// TwinCAT 3 PLC project Untitled1
// ProgramVersion: 3.1.4026.25
// libraries:
//   Tc2_Standard, * (Beckhoff Automation GmbH)
//   Tc2_EtherCAT, * (Beckhoff Automation GmbH)
//   Tc2_System, * (Beckhoff Automation GmbH)
//   Festo_VTEM_DevCon,3.5.7.237,Festo SE & Co. KG
// project tree:
//   / PlcTask.TcTTO
//   POUs/ MAIN.TcPOU, FB_TandemConveyor.TcPOU, FB_CsvDriveSettings.TcPOU
// real-time tasks:
//   TASK PlcTask: cycle T#1ms, priority 20, ADS port 350
// I/O:
//   DEVICE Gerät 1 (EtherCAT), AmsNetId 192.168.178.10.2.1
//     Term 1 (EK1100) [EK1100 EtherCAT Coupler (2A E-Bus)]
//       Term 2 (EL2008) [EL2008 8Ch. Dig. Output 24V, 0.5A]
//       Term 3 (EL2008) [EL2008 8Ch. Dig. Output 24V, 0.5A]
//       Term 4 (EL2004) [EL2004 4Ch. Dig. Output 24V, 0.5A]
//       Term 11 (EL2004) [EL2004 4Ch. Dig. Output 24V, 0.5A]
//       Term 12 (EL1018) [EL1018 8Ch. Dig. Input 24V, 10µs]
//       Term 13 (EL1014-0010) [EL1014-0010 4Ch. Dig. Input 24V, isolated, 10µs]
//       Term 14 (EL3068) [EL3068 8Ch. Ana. Input 0-10V]
//       Term 15 (EL7047) [EL7047 1Ch. Stepper motor output stage (50V, 5A)]
//       Term 22 (EL9011) [EL9011 End Terminal]
//   DEVICE Gerät 2 (EtherCAT), AmsNetId 192.168.178.10.3.1
//     Box 5 (CPX-FB38 64Byte) [CPX-FB38 EtherCAT Busmodul]
//   DEVICE Device 3 (EtherCAT), AmsNetId 10.145.4.14.4.1
//     Term 6 (EK1100) [EK1100 EtherCAT Coupler (2A E-Bus)]
//       Term 7 (EL7201-0010) [EL7201-0010 1Ch. MDP742 Servo motor output stage with OCT (50V, 2.8A RMS)]
//       Term 3 (EL9011) [EL9011 End Terminal]
// variable links:
//   Untitled1/Untitled1 Instance <-> Device 1 (EtherCAT)/Term 1 (EK1100)/Term 11 (EL2004)
//     PlcTask Outputs/MAIN.OpenValve{21..24} <-> Channel {1..4}/Output  (4 links)
//   Untitled1/Untitled1 Instance <-> Device 1 (EtherCAT)/Term 1 (EK1100)/Term 12 (EL1018)
//     PlcTask Inputs/MAIN.LightBarrierOn{1..8} <-> Channel {1..8}/Input  (8 links)
//   Untitled1/Untitled1 Instance <-> Device 1 (EtherCAT)/Term 1 (EK1100)/Term 14 (EL3068)
//     PlcTask Inputs/MAIN.RawNozzlePressure <-> AI Standard Channel 1/Value
//     PlcTask Inputs/MAIN.RawNozzlePressure2 <-> AI Standard Channel 2/Value
//   Untitled1/Untitled1 Instance <-> Device 1 (EtherCAT)/Term 1 (EK1100)/Term 2 (EL2008)
//     PlcTask Outputs/MAIN.OpenValve{1..8} <-> Channel {1..8}/Output  (8 links)
//   Untitled1/Untitled1 Instance <-> Device 1 (EtherCAT)/Term 1 (EK1100)/Term 3 (EL2008)
//     PlcTask Outputs/MAIN.OpenValve{9..16} <-> Channel {1..8}/Output  (8 links)
//   Untitled1/Untitled1 Instance <-> Device 1 (EtherCAT)/Term 1 (EK1100)/Term 4 (EL2004)
//     PlcTask Outputs/MAIN.OpenValve{17..20} <-> Channel {1..4}/Output  (4 links)
//   Untitled1/Untitled1 Instance <-> Device 2 (EtherCAT)/Box 5 (CPX-FB38 64Byte)
//     PlcTask Inputs/MAIN.Valve0_IN[0] @bit 8 <-> Inputs/IB1
//     PlcTask Inputs/MAIN.Valve0_IN[1] @bit 8 <-> Inputs/IB3
//     PlcTask Inputs/MAIN.Valve0_IN[2] @bit 8 <-> Inputs/IB5
//     PlcTask Inputs/MAIN.Valve1_IN[0] @bit 8 <-> Inputs/IB7
//     PlcTask Inputs/MAIN.Valve1_IN[1] @bit 8 <-> Inputs/IB9
//     PlcTask Inputs/MAIN.Valve1_IN[2] @bit 8 <-> Inputs/IB11
//     PlcTask Inputs/MAIN.Valve0_IN[0] <-> Inputs/MAIN.Valve0_IN[0]
//     PlcTask Inputs/MAIN.Valve0_IN[1] <-> Inputs/MAIN.Valve0_IN[1]
//     PlcTask Inputs/MAIN.Valve0_IN[2] <-> Inputs/MAIN.Valve0_IN[2]
//     PlcTask Inputs/MAIN.Valve1_IN[0] <-> Inputs/MAIN.Valve1_IN[0]
//     PlcTask Inputs/MAIN.Valve1_IN[1] <-> Inputs/MAIN.Valve1_IN[1]
//     PlcTask Inputs/MAIN.Valve1_IN[2] <-> Inputs/MAIN.Valve1_IN[2]
//     PlcTask Outputs/MAIN.Valve0_OUT[0] <-> Outputs/MAIN.Valve0_OUT[0]
//     PlcTask Outputs/MAIN.Valve0_OUT[1] <-> Outputs/MAIN.Valve0_OUT[1]
//     PlcTask Outputs/MAIN.Valve0_OUT[2] <-> Outputs/MAIN.Valve0_OUT[2]
//     PlcTask Outputs/MAIN.Valve1_OUT[0] <-> Outputs/MAIN.Valve1_OUT[0]
//     PlcTask Outputs/MAIN.Valve1_OUT[1] <-> Outputs/MAIN.Valve1_OUT[1]
//     PlcTask Outputs/MAIN.Valve1_OUT[2] <-> Outputs/MAIN.Valve1_OUT[2]
//     PlcTask Outputs/MAIN.Valve0_OUT[0] @bit 8 <-> Outputs/QB1
//     PlcTask Outputs/MAIN.Valve0_OUT[1] @bit 8 <-> Outputs/QB3
//     PlcTask Outputs/MAIN.Valve0_OUT[2] @bit 8 <-> Outputs/QB5
//     PlcTask Outputs/MAIN.Valve1_OUT[0] @bit 8 <-> Outputs/QB7
//     PlcTask Outputs/MAIN.Valve1_OUT[1] @bit 8 <-> Outputs/QB9
//     PlcTask Outputs/MAIN.Valve1_OUT[2] @bit 8 <-> Outputs/QB11
//   Untitled1/Untitled1 Instance <-> Device 3 (EtherCAT)/Term 6 (EK1100)/Term 7 (EL7201-0010)
//     PlcTask Inputs/MAIN.ConveyorServo1ActualVelocity <-> DRV Velocity actual value/Velocity actual value
//     PlcTask Inputs/MAIN.ConveyorServo1FeedbackInvalid <-> FB Status/Status/TxPDO State
//     PlcTask Inputs/MAIN.ConveyorServo1InfoState <-> InfoData/State
//     PlcTask Inputs/MAIN.ConveyorServo1Position <-> FB Position/Position
//     PlcTask Inputs/MAIN.ConveyorServo1Statusword <-> DRV Statusword/Statusword
//     PlcTask Inputs/MAIN.ConveyorServo1WcState <-> WcState/WcState
//     PlcTask Outputs/MAIN.ConveyorServo1Controlword <-> DRV Controlword/Controlword
//     PlcTask Outputs/MAIN.ConveyorServo1TargetVelocity <-> DRV Target velocity/Target velocity

CONFIGURATION Untitled1
    RESOURCE PLC ON TwinCAT3
        TASK PlcTask(INTERVAL := T#1ms, PRIORITY := 20);
        PROGRAM MAIN WITH PlcTask : MAIN;
    END_RESOURCE
END_CONFIGURATION

// ---- POUs/MAIN.TcPOU
PROGRAM MAIN
VAR
	State					: INT  := 0; //state machine to control valves and motion terminal
	State2					: INT  := 2; //state machine for nozzle array 2
	State3					: INT  := 0; //state machine for nozzle array 3 and second VTEM unit
	State4					: INT  := 2; //state machine for nozzle array 4
	Counter					: INT  := 0; //timer counter that is in multiples of the PLC task time
	Counter2				: INT  := 0; //timer counter for the second nozzle array
	Counter3				: INT  := 0;
	Counter4				: INT  := 0;
	ShotDurationCycles		: INT  := 100; //100 cycles at 1 ms task time = 100 ms nozzle impulse
	ShotDurationCycles2		: INT  := 100; //pulse duration for the second nozzle array
	ShotDurationCycles3		: INT  := 100;
	ShotDurationCycles4		: INT  := 100;
	DelayDurationCycles		: INT  := 0; //delay cycles at 1 ms task time
	DelayDurationCycles2	: INT  := 0; //delay cycles for the second nozzle array
	DelayDurationCycles3	: INT  := 0;
	DelayDurationCycles4	: INT  := 0;
	OffsetDelayCycles1		: INT  := 0; //velocity-derived delay cycles for the first nozzle array
	OffsetDelayCycles2		: INT  := 0; //velocity-derived delay cycles for the second nozzle array
	OffsetDelayCycles3		: INT  := 0;
	OffsetDelayCycles4		: INT  := 0;
	LatchedDelayCycles1		: INT  := 0;
	LatchedDelayCycles2		: INT  := 0;
	LatchedDelayCycles3		: INT  := 0;
	LatchedDelayCycles4		: INT  := 0;
	LatchedNozzleEndCycles1	: INT  := 100;
	LatchedNozzleEndCycles2	: INT  := 100;
	LatchedNozzleEndCycles3	: INT  := 100;
	LatchedNozzleEndCycles4	: INT  := 100;
	
	TimeDelay				: BOOL := 0;
	DelayCounter			: INT  := 0;
	DelayCounter2			: INT  := 0;
	VelocityTimer			: TON;
	VelocityTimer2			: TON;
	VelocityTimer3			: TON;
	VelocityTimer4			: TON;
	LastVelocityTimeMs		: INT  := 0;
	LastVelocityTime2Ms		: INT  := 0;
	LastVelocityTime3Ms		: INT  := 0;
	LastVelocityTime4Ms		: INT  := 0;
	VelocityTimingActive	: BOOL := FALSE;
	VelocityTiming2Active	: BOOL := FALSE;
	VelocityTiming3Active	: BOOL := FALSE;
	VelocityTiming4Active	: BOOL := FALSE;
	VelocityMeasurementValid: BOOL := FALSE;
	VelocityMeasurement2Valid: BOOL := FALSE;
	VelocityMeasurement3Valid: BOOL := FALSE;
	VelocityMeasurement4Valid: BOOL := FALSE;

	//GUI control values written through ADS
	GuiPressureMbar1		: INT  := 0; // GUI/profile supplies pressure after a PLC restart
	GuiPressureMbar2		: INT  := 0;
	GuiPressureMbar3		: INT  := 0;
	GuiPressureMbar4		: INT  := 0;
	GuiDelayMs1				: UINT := 0;
	GuiDelayMs2				: UINT := 0;
	GuiDelayMs3				: UINT := 0;
	GuiDelayMs4				: UINT := 0;
	GuiPulseDurationMs1		: UINT := 100;
	GuiPulseDurationMs2		: UINT := 100;
	GuiPulseDurationMs3		: UINT := 100;
	GuiPulseDurationMs4		: UINT := 100;
	GuiArrayEnabled1		: BOOL := FALSE; // GUI must explicitly arm nozzle arrays after a PLC restart
	GuiArrayEnabled2		: BOOL := FALSE;
	GuiArrayEnabled3		: BOOL := FALSE;
	GuiArrayEnabled4		: BOOL := FALSE;
	GuiNozzleEnabled1		: BOOL := TRUE;
	GuiNozzleEnabled2		: BOOL := TRUE;
	GuiNozzleEnabled3		: BOOL := TRUE;
	GuiNozzleEnabled4		: BOOL := TRUE;
	GuiNozzleEnabled5		: BOOL := FALSE;
	GuiNozzleEnabled6		: BOOL := FALSE;
	GuiNozzleEnabled7		: BOOL := TRUE;
	GuiNozzleEnabled8		: BOOL := TRUE;
	GuiNozzleEnabled9		: BOOL := TRUE;
	GuiNozzleEnabled10		: BOOL := TRUE;
	GuiNozzleEnabled11		: BOOL := FALSE;
	GuiNozzleEnabled12		: BOOL := FALSE;
	GuiNozzleEnabled13		: BOOL := TRUE;
	GuiNozzleEnabled14		: BOOL := TRUE;
	GuiNozzleEnabled15		: BOOL := TRUE;
	GuiNozzleEnabled16		: BOOL := TRUE;
	GuiNozzleEnabled17		: BOOL := FALSE;
	GuiNozzleEnabled18		: BOOL := FALSE;
	GuiNozzleEnabled19		: BOOL := TRUE;
	GuiNozzleEnabled20		: BOOL := TRUE;
	GuiNozzleEnabled21		: BOOL := TRUE;
	GuiNozzleEnabled22		: BOOL := TRUE;
	GuiNozzleEnabled23		: BOOL := FALSE;
	GuiNozzleEnabled24		: BOOL := FALSE;
	GuiResetVelocityEstimates	: BOOL := FALSE;
	GuiSensorSpacing12Mm	: REAL := 40.0;
	GuiSensorSpacing23Mm	: REAL := 196.0;
	GuiSensorSpacing34Mm	: REAL := 40.0;
	GuiSensorSpacing45Mm	: REAL := 196.0;
	GuiSensorSpacing56Mm	: REAL := 40.0;
	GuiSensorSpacing67Mm	: REAL := 196.0;
	GuiSensorSpacing78Mm	: REAL := 40.0;
	GuiSensor2ToArray1SpacingMm	: REAL := 50.0;
	GuiSensor4ToArray2SpacingMm	: REAL := 45.0;
	GuiSensor6ToArray3SpacingMm	: REAL := 45.0;
	GuiSensor8ToArray4SpacingMm	: REAL := 48.0;
	GuiConveyorEnabled		: BOOL := FALSE;
	GuiVelocityCheckMode	: BOOL := FALSE;
	GuiConveyorReverse		: BOOL := FALSE;
	GuiConveyorReset		: BOOL := FALSE;
	GuiConveyorSpeedMmPerSec	: REAL := 0.0;
	GuiConveyorMaxSpeedMmPerSec	: REAL := 1000.0;
	GuiConveyorCalibrationMode	: BOOL := FALSE;
	GuiCalibrationMarkerDistanceMm	: REAL := 315.0;
	GuiCalibrationJogSteps		: UDINT := 100;
	GuiCalibrationJogSpeedFullStepsPerSec	: REAL := 10.0;
	GuiCalibrationMoveLeft		: BOOL := FALSE;
	GuiCalibrationMoveRight		: BOOL := FALSE;
	GuiCalibrationCaptureLeftMark	: BOOL := FALSE;
	GuiCalibrationCaptureRightMark	: BOOL := FALSE;
	GuiCalibrationStop			: BOOL := FALSE;
	GuiConveyorMmPerFullStep	: REAL := 0.0;
	GuiConveyorCalibrationValid	: BOOL := FALSE;
	// Verified two AM8112 motors, direct drive, 50 mm rollers, same shaft direction.
	// Start remains an explicit GUI command; see CSVSaver/TANDEM_CONVEYOR.md.
	ConveyorServoCommissioned : BOOL := TRUE; // stationary setup and live CoE readback verified; GUI motion starts disabled
	ConveyorServoDirection1 : INT := 1; // same shaft direction, confirmed for the two 50 mm rollers
	ConveyorServoDirection2 : INT := 1;
	ConveyorServoMotor2Ratio : LREAL := 1.0; // motor 2 rev / motor 1 rev, including roller diameter
	ConveyorServoFeedbackCountsPerRev : LREAL := 1048576.0;
	ConveyorServoFeedbackCountsPerRev2 : LREAL := 1048576.0;
	ConveyorServoVelocityUnitsPerRevPerSec : LREAL := 268435.0; // live CoE 0x9010:14 readback
	ConveyorServoVelocityUnitsPerRevPerSec2 : LREAL := 268435.0;
	ConveyorServoMaxMotorRpm : LREAL := 5.0;
	ConveyorServoAccelerationRpmPerSec : LREAL := 5.0;
	ConveyorServoPositionGain : LREAL := 5.0;
	ConveyorServoSyncToleranceFullSteps : LREAL := 5.0;
	ConveyorServoFollowingToleranceFullSteps : LREAL := 20.0;
	// Authoritative NEW belt calibration: 200 virtual full steps per motor 1 revolution.
	// Legacy GUI profiles cannot overwrite this with the old stepper's scale.
	ConveyorServoCalibratedMmPerFullStep : REAL := 0.7853981634; // pi * 50 mm / 200; refine with GUI marker calibration
	ConveyorServoFaultCode : UINT := 0;
	ConveyorServoState : UINT := 0;
	ConveyorServoSyncErrorFullSteps : LREAL := 0.0;
	ConveyorServoStopRequested : BOOL := FALSE;
	ConveyorServoResetRequested : BOOL := FALSE;
	TandemConveyor : FB_TandemConveyor;
	ConveyorDriveSettings : FB_CsvDriveSettings;
	GuiOffsetMm1			: REAL := 0.0;
	GuiOffsetMm2			: REAL := 0.0;
	GuiOffsetMm3			: REAL := 0.0;
	GuiOffsetMm4			: REAL := 0.0;
	GuiForceDelayMeasurementEnabled	: BOOL := FALSE;
	GuiForceDelayLightBarrier	: UINT := 2;
	GuiForceDelaySensor		: UINT := 1;
	GuiForceDelayWindowMs		: UINT := 2000;
	GuiForceDelayMinRise		: REAL := 0.05;
	GuiForceDelayReset		: BOOL := FALSE;
	GuiForceResponseDelayMs1	: REAL := 8.7;
	GuiForceResponseDelayMs2	: REAL := 8.7;
	GuiForceResponseDelayMs3	: REAL := 8.7;
	GuiForceResponseDelayMs4	: REAL := 8.7;
	GuiForceSingleNozzleResponseDelayMs1	: REAL := 8.7;
	GuiForceSingleNozzleResponseDelayMs2	: REAL := 8.7;
	GuiForceSingleNozzleResponseDelayMs3	: REAL := 8.7;
	GuiForceSingleNozzleResponseDelayMs4	: REAL := 8.7;
	// BiBaZu Reorientation Control ADS contract
	GuiReorientationControlActive	: BOOL := FALSE;
	GuiReorientationHeartbeat		: UDINT := 0;
	GuiReorientationStart			: BOOL := FALSE;
	GuiReorientationAbort			: BOOL := FALSE;
	GuiReorientationReset			: BOOL := FALSE;
	GuiReorientationLegacyTakeover	: BOOL := FALSE;
	GuiReorientationExpectedArrayMask	: BYTE := 0;
	// Continuous production-run staging area.  The GUI writes every field first
	// and publishes it atomically by incrementing QueueCommit last.
	GuiReorientationFinish			: BOOL := FALSE;
	GuiReorientationResultAck		: UDINT := 0;
	GuiReorientationQueueCommit		: UDINT := 0;
	GuiReorientationQueueSequence	: UDINT := 0;
	GuiReorientationQueueTrackId		: UDINT := 0;
	GuiReorientationQueuePoseId		: UINT := 0;
	GuiReorientationQueueDecisionCode	: UINT := 0;
	GuiReorientationQueueArrayMask	: BYTE := 0;
	GuiReorientationQueueNozzleMask1	: BYTE := 0;
	GuiReorientationQueueNozzleMask2	: BYTE := 0;
	GuiReorientationQueueNozzleMask3	: BYTE := 0;
	GuiReorientationQueueNozzleMask4	: BYTE := 0;
	GuiReorientationQueuePressureMbar1	: INT := 0;
	GuiReorientationQueuePressureMbar2	: INT := 0;
	GuiReorientationQueuePressureMbar3	: INT := 0;
	GuiReorientationQueuePressureMbar4	: INT := 0;
	GuiReorientationQueueDelayMs1	: UINT := 0;
	GuiReorientationQueueDelayMs2	: UINT := 0;
	GuiReorientationQueueDelayMs3	: UINT := 0;
	GuiReorientationQueueDelayMs4	: UINT := 0;
	GuiReorientationQueuePulseMs1	: UINT := 1;
	GuiReorientationQueuePulseMs2	: UINT := 1;
	GuiReorientationQueuePulseMs3	: UINT := 1;
	GuiReorientationQueuePulseMs4	: UINT := 1;
	GuiReorientationQueueOffsetMm1	: REAL := 0.0;
	GuiReorientationQueueOffsetMm2	: REAL := 0.0;
	GuiReorientationQueueOffsetMm3	: REAL := 0.0;
	GuiReorientationQueueOffsetMm4	: REAL := 0.0;
	GuiReorientationQueueForceResponseMs1	: REAL := 0.0;
	GuiReorientationQueueForceResponseMs2	: REAL := 0.0;
	GuiReorientationQueueForceResponseMs3	: REAL := 0.0;
	GuiReorientationQueueForceResponseMs4	: REAL := 0.0;
	GuiReorientationQueueForceSingleMs1	: REAL := 0.0;
	GuiReorientationQueueForceSingleMs2	: REAL := 0.0;
	GuiReorientationQueueForceSingleMs3	: REAL := 0.0;
	GuiReorientationQueueForceSingleMs4	: REAL := 0.0;
	ReorientationHeartbeatAck		: UDINT := 0;
	ReorientationHeartbeatAlive	: BOOL := FALSE;
	ReorientationState				: UINT := 0; //0 legacy,10 armed,20 running,30 drain,40 complete,90+ fault
	ReorientationFaultCode			: UINT := 0;
	ReorientationBusy				: BOOL := FALSE;
	ReorientationExitSeen			: BOOL := FALSE;
	ReorientationArraysIdle		: BOOL := TRUE;
	ReorientationExpectedArrayMask	: BYTE := 0;
	ReorientationTriggeredArrayMask	: BYTE := 0;
	ReorientationComplete			: BOOL := FALSE;
	ReorientationCycleCounter		: UDINT := 0;
	ReorientationLastHeartbeat		: UDINT := 0;
	ReorientationHeartbeatAgeMs	: UDINT := 0;
	ReorientationCycleAgeMs		: UDINT := 0;
	ReorientationDrainAgeMs		: UDINT := 0;
	ReorientationSafeLatch			: BOOL := FALSE;
	// Diagnostic context retained for non-fatal light-barrier warnings and for
	// compatibility with older GUIs that reported these conditions as fault 96.
	ReorientationFaultDetail		: UINT := 0; // 1=no clear, 2=queue mismatch, 3=sensor order
	ReorientationFaultSensor		: UINT := 0;
	ReorientationFaultExpectedSequence	: UDINT := 0;
	ReorientationFaultPreviousSequence	: UDINT := 0;
	ReorientationFaultQueueAck		: UDINT := 0;
	ReorientationFaultQueueSlotSequence	: UDINT := 0;
	ReorientationFaultBarrierStableMask	: BYTE := 0;
	// Non-fatal resynchronization after an intentionally airborne workpiece
	// skips barriers downstream of its final active nozzle array.
	// 1=downstream barriers skipped, 2=airborne duplicate, 3=no-clear edge,
	// 4=edge without matching queue slot, 5=out-of-order edge. All are non-fatal.
	ReorientationWarningCode		: UINT := 0;
	ReorientationWarningSensor		: UINT := 0;
	ReorientationWarningSequence	: UDINT := 0;
	ReorientationWarningPreviousSequence	: UDINT := 0;
	ReorientationWarningSkippedBarrierMask	: BYTE := 0;
	ReorientationWarningCounter		: UDINT := 0;
	// Public continuous-run queue/result diagnostics.
	ReorientationQueueDepth			: UINT := 0;
	ReorientationQueueCapacity		: UINT := 128;
	ReorientationQueueEnqueueAck		: UDINT := 0;
	ReorientationQueueEnteredCount	: UDINT := 0;
	ReorientationQueueCompletedCount	: UDINT := 0;
	ReorientationQueueBypassCount		: UDINT := 0;
	ReorientationSensorSequence1	: UDINT := 0;
	ReorientationSensorSequence2	: UDINT := 0;
	ReorientationSensorSequence3	: UDINT := 0;
	ReorientationSensorSequence4	: UDINT := 0;
	ReorientationSensorSequence5	: UDINT := 0;
	ReorientationSensorSequence6	: UDINT := 0;
	ReorientationSensorSequence7	: UDINT := 0;
	ReorientationSensorSequence8	: UDINT := 0;
	ReorientationResultAvailable	: BOOL := FALSE;
	ReorientationResultSequence		: UDINT := 0;
	ReorientationResultTriggeredMask	: BYTE := 0;
	ReorientationResultFaultCode	: UINT := 0;
	// Frozen 128-part ring.  A slot is not reusable until its result is ACKed.
	BatchQueueSequence				: ARRAY [0..127] OF UDINT;
	BatchQueueTrackId				: ARRAY [0..127] OF UDINT;
	BatchQueuePoseId				: ARRAY [0..127] OF UINT;
	BatchQueueDecisionCode			: ARRAY [0..127] OF UINT;
	BatchQueueArrayMask				: ARRAY [0..127] OF BYTE;
	BatchQueueNozzleMask			: ARRAY [0..127, 1..4] OF BYTE;
	BatchQueuePressureMbar			: ARRAY [0..127, 1..4] OF INT;
	BatchQueueDelayMs				: ARRAY [0..127, 1..4] OF UINT;
	BatchQueuePulseMs				: ARRAY [0..127, 1..4] OF UINT;
	BatchQueueOffsetMm				: ARRAY [0..127, 1..4] OF REAL;
	BatchQueueForceResponseMs		: ARRAY [0..127, 1..4] OF REAL;
	BatchQueueForceSingleMs			: ARRAY [0..127, 1..4] OF REAL;
	BatchQueuePairStartMs			: ARRAY [0..127, 1..4] OF UDINT;
	BatchQueueTriggeredMask			: ARRAY [0..127] OF BYTE;
	// Unlike TriggeredMask, this is set only while a real valve output is
	// commanded open. It marks this exact queued part as eligible for flight
	// recovery; it cannot prove pneumatic pressure or actual part motion.
	BatchQueueActuatedMask			: ARRAY [0..127] OF BYTE;
	BatchQueueFinishedMask			: ARRAY [0..127] OF BYTE;
	BatchQueueExitSeen				: ARRAY [0..127] OF BOOL;
	BatchResultSequence				: ARRAY [0..127] OF UDINT;
	BatchResultTriggeredMask		: ARRAY [0..127] OF BYTE;
	BatchResultFaultCode			: ARRAY [0..127] OF UINT;
	BatchNextSensorSequence			: ARRAY [1..8] OF UDINT;
	BatchSensorSequence				: ARRAY [1..8] OF UDINT;
	BatchSensorFalling				: ARRAY [1..8] OF BOOL;
	BatchSensorStable				: ARRAY [1..8] OF BOOL;
	BatchPairSpacingMm				: ARRAY [1..4] OF REAL;
	BatchSensorToArraySpacingMm	: ARRAY [1..4] OF REAL;
	BatchSensorNeedsClear			: ARRAY [1..8] OF BOOL;
	PairedFirstBarrierFalling		: ARRAY [1..4] OF BOOL;
	PairedFirstBarrierLocked		: ARRAY [1..4] OF BOOL;
	PairedFirstBarrierLockStartMs	: ARRAY [1..4] OF UDINT;
	PairedSecondBarrierFalling		: ARRAY [1..4] OF BOOL;
	PairedSecondBarrierLocked		: ARRAY [1..4] OF BOOL;
	PairedSecondBarrierLockStartMs	: ARRAY [1..4] OF UDINT;
	PairedBarrierLockTimeoutMs		: UDINT := 500;
	BatchSensorOrderInvalid			: BOOL := FALSE;
	BatchCanResyncSkippedSensors	: BOOL := FALSE;
	BatchCurrentFlightConfirmed	: BOOL := FALSE;
	BatchIgnoreAirborneDuplicate	: BOOL := FALSE;
	BatchLastRequiredSensor			: INT := 0;
	BatchLastRequiredArrayMask		: BYTE := 0;
	BatchPreviousSlotIndex			: INT := 0;
	BatchPreviousLastRequiredSensor	: INT := 0;
	BatchPreviousLastRequiredArrayMask	: BYTE := 0;
	BatchResyncIndex					: INT := 0;
	BatchSkippedBarrierMask			: BYTE := 0;
	BatchCurrentBarrierStableMask	: BYTE := 0;
	BatchNextCompleteSequence		: UDINT := 1;
	BatchLastAcceptedCommit			: UDINT := 0;
	BatchAcceptedResultAck			: UDINT := 0;
	// Each array has its own 16-entry job FIFO.  Jobs contain the final delay,
	// pressure and nozzle mask and therefore remain immutable during a pulse.
	BatchJobSequence				: ARRAY [0..15, 1..4] OF UDINT;
	BatchJobNozzleMask				: ARRAY [0..15, 1..4] OF BYTE;
	BatchJobPressureMbar			: ARRAY [0..15, 1..4] OF INT;
	BatchJobDelayCycles				: ARRAY [0..15, 1..4] OF INT;
	BatchJobPulseCycles				: ARRAY [0..15, 1..4] OF INT;
	BatchJobHead					: ARRAY [1..4] OF UINT;
	BatchJobTail					: ARRAY [1..4] OF UINT;
	BatchJobCount					: ARRAY [1..4] OF UINT;
	BatchActiveSequence				: ARRAY [1..4] OF UDINT;
	BatchLoopIndex					: INT := 0;
	BatchSlotIndex					: INT := 0;
	BatchJobIndex					: INT := 0;
	BatchElapsedMs					: UDINT := 0;
	BatchComputedDelayMs			: REAL := 0.0;
	BatchResponseDelayMs			: REAL := 0.0;
	BatchNozzleCount				: INT := 0;
	EstimatedVelocityMmPerSec	: REAL := 0.0;
	EstimatedVelocityMmPerSec1	: REAL := 0.0;
	EstimatedVelocityMmPerSec2	: REAL := 0.0;
	EstimatedVelocityMmPerSec3	: REAL := 0.0;
	EstimatedVelocityMmPerSec4	: REAL := 0.0;
	EstimatedOffsetDelayMs1		: REAL := 0.0;
	EstimatedOffsetDelayMs2		: REAL := 0.0;
	EstimatedOffsetDelayMs3		: REAL := 0.0;
	EstimatedOffsetDelayMs4		: REAL := 0.0;
	Array1Active			: BOOL := FALSE;
	Array2Active			: BOOL := FALSE;
	Array3Active			: BOOL := FALSE;
	Array4Active			: BOOL := FALSE;
	ConveyorSpeedMmPerSec	: REAL := 0.0; //limited conveyor speed command in mm/s
	ConveyorVelocityRatio	: REAL := 0.0;
	ConveyorVelocityRaw		: INT := 0; //0..10000 legacy velocity command, adapted to both servos
	ConveyorFullStepsPerSec	: REAL := 0.0;
	ConveyorSpeedRangeFullStepsPerSec	: REAL := 2000.0; //legacy velocity scale, virtual full steps/s
	ConveyorMotionState		: INT := 0;
	ConveyorMotionMode		: INT := 0; //0 idle, 1 normal endless, 2 calibration move
	ConveyorActiveVelocity	: INT := 0;
	ConveyorActiveStartType	: UINT := 0;
	CalibrationTargetIncrements	: DINT := 0;
	CalibrationDirectionNegative	: BOOL := FALSE;
	CalibrationLeftMarkValid	: BOOL := FALSE;
	CalibrationRightMarkValid	: BOOL := FALSE;
	CalibrationLeftPosition		: UDINT := 0;
	CalibrationRightPosition	: UDINT := 0;
	CalibrationPositionDifferenceIncrements	: UDINT := 0;
	CalibrationFullStepDifference	: REAL := 0.0;
	CalibrationStepsPerMm		: REAL := 0.0;
	CalibrationBusy			: BOOL := FALSE;
	CalibrationError			: BOOL := FALSE;
	CalibrationStatusCode		: UINT := 0; //0 ready, 1 starting, 2 moving, 3 complete, 4 invalid, 5 drive error
	CalibrationPositionDelta	: LINT := 0;
	LastConveyorCalibrationMode	: BOOL := FALSE;
	GuiBarrierCalibrationFirstSensor	: UINT := 1;
	GuiBarrierCalibrationSecondSensor	: UINT := 2;
	GuiBarrierCalibrationDebounceMs	: UINT := 20;
	GuiLightBarrierInvert1	: BOOL := TRUE;
	GuiLightBarrierInvert2	: BOOL := TRUE;
	GuiLightBarrierInvert3	: BOOL := TRUE;
	GuiLightBarrierInvert4	: BOOL := TRUE;
	GuiLightBarrierInvert5	: BOOL := TRUE;
	GuiLightBarrierInvert6	: BOOL := TRUE;
	GuiLightBarrierInvert7	: BOOL := TRUE;
	GuiLightBarrierInvert8	: BOOL := TRUE;
	GuiLightBarrierDebounceEnabled1	: BOOL := FALSE;
	GuiLightBarrierDebounceEnabled2	: BOOL := FALSE;
	GuiLightBarrierDebounceEnabled3	: BOOL := FALSE;
	GuiLightBarrierDebounceEnabled4	: BOOL := FALSE;
	GuiLightBarrierDebounceEnabled5	: BOOL := FALSE;
	GuiLightBarrierDebounceEnabled6	: BOOL := FALSE;
	GuiLightBarrierDebounceEnabled7	: BOOL := FALSE;
	GuiLightBarrierDebounceEnabled8	: BOOL := FALSE;
	GuiBarrierCalibrationStart	: BOOL := FALSE;
	BarrierCalibrationActive	: BOOL := FALSE;
	BarrierCalibrationFirstCaptured	: BOOL := FALSE;
	BarrierCalibrationSecondCaptured	: BOOL := FALSE;
	BarrierCalibrationValid	: BOOL := FALSE;
	BarrierCalibrationFirstPosition	: UDINT := 0;
	BarrierCalibrationSecondPosition	: UDINT := 0;
	BarrierCalibrationDifferenceIncrements	: UDINT := 0;
	BarrierCalibrationDistanceMm	: REAL := 0.0;
	BarrierCalibrationPositionDelta	: LINT := 0;
	BarrierCalibrationFirstState	: BOOL := FALSE;
	BarrierCalibrationSecondState	: BOOL := FALSE;
	BarrierCalibrationFirstInitialState	: BOOL := FALSE;
	BarrierCalibrationSecondInitialState	: BOOL := FALSE;
	BarrierCalibrationFirstCandidatePosition	: UDINT := 0;
	BarrierCalibrationSecondCandidatePosition	: UDINT := 0;
	BarrierCalibrationFirstStableCycles	: UINT := 0;
	BarrierCalibrationSecondStableCycles	: UINT := 0;
	BarrierCalibrationAbortRequested	: BOOL := FALSE;
	BarrierCalibrationStatusCode	: UINT := 0; //0 ready, 1 waiting first, 2 waiting second, 3 complete, 4 invalid/cancelled, 5 drive error

	//IO Variables
	//EL 1018
	LightBarrierOn1 AT %I*	: BOOL := 0; //1 when detecting a reflection
	LightBarrierOn2 AT %I*	: BOOL := 0; //1 when detecting a reflection
	LightBarrierOn3 AT %I*	: BOOL := 0; //1 when detecting a reflection
	LightBarrierOn4 AT %I*	: BOOL := 0; //1 when detecting a reflection
	LightBarrierOn5 AT %I*	: BOOL := 0; //1 when detecting a reflection
	LightBarrierOn6 AT %I*	: BOOL := 0; //1 when detecting a reflection
	LightBarrierOn7 AT %I*	: BOOL := 0; //1 when detecting a reflection
	LightBarrierOn8 AT %I*	: BOOL := 0; //1 when detecting a reflection
	LightBarrierLogical1	: BOOL := FALSE;
	LightBarrierLogical2	: BOOL := FALSE;
	LightBarrierLogical3	: BOOL := FALSE;
	LightBarrierLogical4	: BOOL := FALSE;
	LightBarrierLogical5	: BOOL := FALSE;
	LightBarrierLogical6	: BOOL := FALSE;
	LightBarrierLogical7	: BOOL := FALSE;
	LightBarrierLogical8	: BOOL := FALSE;
	LastLightBarrierInvert1	: BOOL := FALSE;
	LastLightBarrierInvert2	: BOOL := FALSE;
	LastLightBarrierInvert3	: BOOL := TRUE;
	LastLightBarrierInvert4	: BOOL := TRUE;
	LastLightBarrierInvert5	: BOOL := FALSE;
	LastLightBarrierInvert6	: BOOL := FALSE;
	LastLightBarrierInvert7	: BOOL := TRUE;
	LastLightBarrierInvert8	: BOOL := TRUE;
	LastLightBarrierDebounceEnabled1	: BOOL := TRUE;
	LastLightBarrierDebounceEnabled2	: BOOL := TRUE;
	LastLightBarrierDebounceEnabled3	: BOOL := FALSE;
	LastLightBarrierDebounceEnabled4	: BOOL := FALSE;
	LastLightBarrierDebounceEnabled5	: BOOL := TRUE;
	LastLightBarrierDebounceEnabled6	: BOOL := TRUE;
	LastLightBarrierDebounceEnabled7	: BOOL := FALSE;
	LastLightBarrierDebounceEnabled8	: BOOL := FALSE;
	LightBarrierStable1		: BOOL := FALSE;
	LightBarrierStable2		: BOOL := FALSE;
	LightBarrierStable3		: BOOL := FALSE;
	LightBarrierStable4		: BOOL := FALSE;
	LightBarrierStable5		: BOOL := FALSE;
	LightBarrierStable6		: BOOL := FALSE;
	LightBarrierStable7		: BOOL := FALSE;
	LightBarrierStable8		: BOOL := FALSE;
	LightBarrierStableCounter1	: UINT := 0;
	LightBarrierStableCounter2	: UINT := 0;
	LightBarrierStableCounter3	: UINT := 0;
	LightBarrierStableCounter4	: UINT := 0;
	LightBarrierStableCounter5	: UINT := 0;
	LightBarrierStableCounter6	: UINT := 0;
	LightBarrierStableCounter7	: UINT := 0;
	LightBarrierStableCounter8	: UINT := 0;
	LightBarrierDebounceInitialized	: BOOL := FALSE;
	LastLightBarrier1		: BOOL := FALSE; //previous debounced state
	LastLightBarrier2		: BOOL := FALSE; //previous debounced state
	LastLightBarrier3		: BOOL := FALSE; //previous debounced state
	LastLightBarrier4		: BOOL := FALSE; //previous debounced state
	LastLightBarrier5		: BOOL := FALSE; //previous debounced state
	LastLightBarrier6		: BOOL := FALSE; //previous debounced state
	LastLightBarrier7		: BOOL := FALSE; //previous debounced state
	LastLightBarrier8		: BOOL := FALSE; //previous debounced state
	LightBarrier1FallingEdge	: BOOL := FALSE;
	LightBarrier2FallingEdge	: BOOL := FALSE;
	LightBarrier3FallingEdge	: BOOL := FALSE;
	LightBarrier4FallingEdge	: BOOL := FALSE;
	LightBarrier5FallingEdge	: BOOL := FALSE;
	LightBarrier6FallingEdge	: BOOL := FALSE;
	LightBarrier7FallingEdge	: BOOL := FALSE;
	LightBarrier8FallingEdge	: BOOL := FALSE;
	LightBarrierEventClockMs	: UDINT := 0; //1 ms PLC task cycle counter
	// ADS diagnostic ring: version, sequence, clock, then 256 records
	// (sequence, timestamp_ms, sensor * 2 + stable_state). Never consumed by ADS.
	LightBarrierEventHistory : ARRAY[0..770] OF UDINT;
	LightBarrierHistorySlot : UDINT := 0;
	// Actual alternating-gate outputs used by velocity timing and array triggers.
	// Same ring layout, but code bit 0 is the accepted-edge BOOL (1 for one cycle).
	LightBarrierFilteredEventHistory : ARRAY[0..770] OF UDINT;
	LightBarrierFilteredSignal : ARRAY[1..8] OF BOOL;
	LastLightBarrierFilteredSignal : ARRAY[1..8] OF BOOL;
	LightBarrierFilteredSensor : INT;
	LightBarrierFilteredSlot : UDINT;
	LightBarrierEventCount1	: UDINT := 0;
	LightBarrierEventCount2	: UDINT := 0;
	LightBarrierEventCount3	: UDINT := 0;
	LightBarrierEventCount4	: UDINT := 0;
	LightBarrierEventCount5	: UDINT := 0;
	LightBarrierEventCount6	: UDINT := 0;
	LightBarrierEventCount7	: UDINT := 0;
	LightBarrierEventCount8	: UDINT := 0;
	LightBarrierLastEventTimeMs1	: UDINT := 0;
	LightBarrierLastEventTimeMs2	: UDINT := 0;
	LightBarrierLastEventTimeMs3	: UDINT := 0;
	LightBarrierLastEventTimeMs4	: UDINT := 0;
	LightBarrierLastEventTimeMs5	: UDINT := 0;
	LightBarrierLastEventTimeMs6	: UDINT := 0;
	LightBarrierLastEventTimeMs7	: UDINT := 0;
	LightBarrierLastEventTimeMs8	: UDINT := 0;
	LightBarrierLastEventPosition1	: UDINT := 0;
	LightBarrierLastEventPosition2	: UDINT := 0;
	LightBarrierLastEventPosition3	: UDINT := 0;
	LightBarrierLastEventPosition4	: UDINT := 0;
	LightBarrierLastEventPosition5	: UDINT := 0;
	LightBarrierLastEventPosition6	: UDINT := 0;
	LightBarrierLastEventPosition7	: UDINT := 0;
	LightBarrierLastEventPosition8	: UDINT := 0;
	Array1TriggerPending		: BOOL := FALSE;
	Array2TriggerPending		: BOOL := FALSE;
	Array3TriggerPending		: BOOL := FALSE;
	Array4TriggerPending		: BOOL := FALSE;
	ForceDelayBusy			: BOOL := FALSE;
	ForceDelayStatusCode		: UINT := 0; //0 disabled, 1 armed, 2 measuring, 3 valid, 4 no peak
	ForceDelayResultCounter		: UDINT := 0;
	ForceDelayValidCount		: UDINT := 0;
	ForceDelayInvalidCount		: UDINT := 0;
	ForceDelayLastValid		: BOOL := FALSE;
	ForceDelayLightBarrierTimeMs	: UDINT := 0;
	ForceDelayPeakTimeMs		: UDINT := 0;
	ForceDelayPeakDelayMs		: UDINT := 0;
	ForceDelayElapsedMs		: UINT := 0;
	ForceDelayBaseline		: REAL := 0.0;
	ForceDelayPeak			: REAL := 0.0;
	ForceDelayPeakRise		: REAL := 0.0;
	ForceDelayCurrentSignal		: REAL := 0.0;
	ForceDelayBaselineBuffer1	: ARRAY [0..49] OF REAL;
	ForceDelayBaselineBuffer2	: ARRAY [0..49] OF REAL;
	ForceDelayBaselineSum1		: REAL := 0.0;
	ForceDelayBaselineSum2		: REAL := 0.0;
	ForceDelayBaselineIndex		: UINT := 0;
	ForceDelayBaselineCount		: UINT := 0;
	ForceDelayTrigger		: BOOL := FALSE;
	ActiveNozzleCount1		: INT := 0;
	ActiveNozzleCount2		: INT := 0;
	ActiveNozzleCount3		: INT := 0;
	ActiveNozzleCount4		: INT := 0;
	EffectiveForceResponseDelayMs1	: REAL := 0.0;
	EffectiveForceResponseDelayMs2	: REAL := 0.0;
	EffectiveForceResponseDelayMs3	: REAL := 0.0;
	EffectiveForceResponseDelayMs4	: REAL := 0.0;
	
	//EL 3068
	RawNozzlePressure AT %I*: INT  := 0; //The raw analogue input reading from the EL3068 terminal (max 32767)
	NozzlePressure			: REAL := 0.0; //converted to pressure value in bar
	
	RawNozzlePressure2 AT %I*: INT := 0; //raw reading from the second pressure sensor
	NozzlePressure2          : REAL := 0.0; //converted to pressure value in bar
	
	
	//Digital valve outputs
	//0 to close valve 1 to open valve
	OpenValve1 AT %Q*		: BOOL := 0;
	OpenValve2 AT %Q*		: BOOL := 0;
	OpenValve3 AT %Q*		: BOOL := 0;
	OpenValve4 AT %Q*		: BOOL := 0;
	OpenValve5 AT %Q*		: BOOL := 0;
	OpenValve6 AT %Q*		: BOOL := 0;
	OpenValve7 AT %Q*		: BOOL := 0;
	OpenValve8 AT %Q*		: BOOL := 0;
	OpenValve9 AT %Q*		: BOOL := 0;
	OpenValve10 AT %Q*		: BOOL := 0;
	OpenValve11 AT %Q*		: BOOL := 0;
	OpenValve12 AT %Q*		: BOOL := 0;
	OpenValve13 AT %Q*		: BOOL := 0;
	OpenValve14 AT %Q*		: BOOL := 0;
	OpenValve15 AT %Q*		: BOOL := 0;
	OpenValve16 AT %Q*		: BOOL := 0;
	OpenValve17 AT %Q*		: BOOL := 0;
	OpenValve18 AT %Q*		: BOOL := 0;
	OpenValve19 AT %Q*		: BOOL := 0;
	OpenValve20 AT %Q*		: BOOL := 0;
	OpenValve21 AT %Q*		: BOOL := 0;
	OpenValve22 AT %Q*		: BOOL := 0;
	OpenValve23 AT %Q*		: BOOL := 0;
	OpenValve24 AT %Q*		: BOOL := 0;

	// Existing ADS contract, now backed by FB_TandemConveyor rather than EL7047 I/O.
	StepperStmStatus : WORD := 0;
	StepperPosBusy : BOOL := FALSE;
	StepperPosInTarget : BOOL := FALSE;
	StepperPosWarning : BOOL := FALSE;
	StepperPosError : BOOL := FALSE;
	StepperPosReadyToExecute : BOOL := FALSE;
	StepperInternalPosition : UDINT := 0; // encoder feedback, 64 increments per virtual full step
	StepperWcState : BOOL := TRUE;
	StepperInfoDataState : UINT := 0;
	StepperControlEnable : BOOL := FALSE;
	StepperControlReset : BOOL := FALSE;
	StepperControlReduceTorque : BOOL := FALSE;
	StepperControlDigitalOutput1 : BOOL := FALSE;
	StepperPosExecute : BOOL := FALSE;
	StepperPosEmergencyStop : BOOL := FALSE;
	StepperPosTargetPosition : UDINT := 0;
	StepperPosVelocity : INT := 0;
	StepperPosStartType : UINT := 0;
	StepperPosAcceleration : UINT := 1000; // compatibility only; servo ramp configured above
	StepperPosDeceleration : UINT := 1000;
	// Two EL7201-0010 terminals; mapped to the same 1 ms task.
	ConveyorServo1Position AT %I* : UDINT;
	ConveyorServo1Statusword AT %I* : UINT;
	ConveyorServo1ActualVelocity AT %I* : DINT;
	ConveyorServo1FeedbackInvalid AT %I* : BOOL := TRUE;
	ConveyorServo1WcState AT %I* : BOOL := TRUE;
	ConveyorServo1InfoState AT %I* : UINT;
	ConveyorServo1Controlword AT %Q* : UINT;
	ConveyorServo1TargetVelocity AT %Q* : DINT;
	ConveyorServo2Position : UDINT;
	ConveyorServo2Statusword : UINT;
	ConveyorServo2ActualVelocity : DINT;
	ConveyorServo2FeedbackInvalid : BOOL := TRUE;
	ConveyorServo2WcState : BOOL := TRUE;
	ConveyorServo2InfoState : UINT;
	ConveyorServo2Controlword : UINT;
	ConveyorServo2TargetVelocity : DINT;
	
	//VTEM Motion Terminal Variables
	FBValveControlV0		: FestoVTEMdc.FB_ValveControl; //Renaming function in program
	Valve0_IN AT %I*		: ARRAY [0..2] OF WORD;			//Input for VTEM Valves
	Valve0_OUT AT %Q*		: ARRAY [0..2] OF WORD;			//Output for VTEM Valves starts at QB0 and increases by 6 for every sequential insel
	Enable0					: BOOL := FALSE;				//Enables VTEM Valves
	Acknowledge0			: BOOL := FALSE;				//Acknowledges the Enabling variable. Must be done after enable is set to true
	ValveMode0				: BYTE := 3;					//Motion app used
	AppControl0				: BYTE := 3;					//0 = no valves, 1 = Valve02 only, 2 = valve04 only, 3 = both valves
	AppOption0				: BYTE;							//only used for motion apps 1 and 2
	PresValueV02			: INT  := 0;					//set pressure for V02 in thousandths of bar (1000 = 1 bar)
	PresValueV04			: INT  := 0;					//set pressure for V04
	ActValveMode0			: BYTE;							
	ActValveState0			: BYTE;
	ActAppState0			: INT;
	ActPresValueV02			: INT;							//Actual pressure output for V02
	ActPresValueV04			: INT;							//Actual pressure output for V04
	ResponseToValveModeSet0	: INT;							//Gives status of VTEM Terminal
	ErrorCode0				: INT;							//Must = 0, otherwise lookup errorcode

	FBValveControlV1		: FestoVTEMdc.FB_ValveControl; //Pressure control for VTEM unit 1
	Valve1_IN AT %I*		: ARRAY [0..2] OF WORD;			//Input for VTEM unit 1 valves
	Valve1_OUT AT %Q*		: ARRAY [0..2] OF WORD;			//Output for VTEM unit 1 valves, link to the next 6-byte insel
	Enable1					: BOOL := FALSE;				//Enables VTEM unit 1 valves
	Acknowledge1			: BOOL := FALSE;				//Acknowledges unit 1 enabling variable
	ValveMode1				: BYTE := 3;					//Motion app used
	AppControl1				: BYTE := 3;					//0 = no valves, 1 = Valve02 only, 2 = valve04 only, 3 = both valves
	AppOption1				: BYTE;							//only used for motion apps 1 and 2
	PresValueV12			: INT := 0;						//set pressure for unit 1 V02, used by nozzle array 3
	PresValueV14			: INT := 0;						//set pressure for unit 1 V04, used by nozzle array 4
	ActValveMode1			: BYTE;
	ActValveState1			: BYTE;
	ActAppState1			: INT;
	ActPresValueV12			: INT;							//Actual pressure output for unit 1 V02
	ActPresValueV14			: INT;							//Actual pressure output for unit 1 V04
	ResponseToValveModeSet1	: INT;							//Gives status of VTEM unit 1
	ErrorCode1				: INT;							//Must = 0, otherwise lookup errorcode
	
	//Pressure Variables
	PressureSum             : REAL  := 0.0;                 //sum of data points recorded by pressure sensor
	PressurePoints          : INT   := 0;                   //value for number of data points recorded by pressure sensor	
	PressureSum1            : REAL  := 0.0;                 //sum of pressure from nozzle 1
	PressureSum2            : REAL  := 0.0;                 //sum of pressure from nozzle 2
	PressurePoints1         : INT   := 0;
	PressurePoints2         : INT   := 0;
	
	AvgPressure             : REAL  := 0.0;                 //average pressure between the two nozzles
	AvgPressureN1           : REAL  := 0.0;                 //average pressure of the first nozzle
	AvgPressureN2           : REAL  := 0.0;                 //average pressure of the second nozzle 
	ShotCounter				: UDINT := 0;					//increments once for every completed nozzle shot
	LogPressureTrigger		: BOOL  := FALSE;				//one PLC-cycle pulse when a new shot value is ready
	
	N1PressureValues        : ARRAY [0..1000] OF REAL;        //array for the output of pressure values for nozzle 1
	N2PressureValues        : ARRAY [0..1000] OF REAL;        //array for the ouput of pressure values for nozzle 2

	NozzlePressures         : ARRAY [0..1000, 0..1] OF REAL;

END_VAR

// Preserve commands before the legacy state machine consumes their one-shot flags.
ConveyorServoStopRequested := GuiCalibrationStop;
ConveyorServoResetRequested := GuiConveyorReset;
// Profiles for the old belt must not silently replace the new belt's calibration.
GuiConveyorMmPerFullStep := ConveyorServoCalibratedMmPerFullStep;
GuiConveyorCalibrationValid := ConveyorServoCalibratedMmPerFullStep > 0.0;
IF NOT ConveyorServoCommissioned OR NOT GuiConveyorCalibrationValid THEN
	GuiConveyorEnabled := FALSE;
END_IF
// Surface current-cycle drive/communication faults before the batch safety checks.
ConveyorDriveSettings(Online := (ConveyorServo1InfoState = 8) AND NOT ConveyorServo1WcState);
StepperWcState := ConveyorServo1WcState;
StepperInfoDataState := ConveyorServo1InfoState;

StepperPosError := TandemConveyor.Error OR (ConveyorServoCommissioned AND (
	((ConveyorServo1Statusword AND UINT#8) <> 0)
	OR StepperWcState OR (StepperInfoDataState <> UINT#8)
	OR ConveyorServo1FeedbackInvalid OR NOT ConveyorDriveSettings.Valid));

NozzlePressure := TO_REAL(RawNozzlePressure) * 10.0 / 32767.0;
NozzlePressure2 := TO_REAL(RawNozzlePressure2) * 10.0 / 32767.0;
LogPressureTrigger := FALSE;
LightBarrierEventClockMs := LightBarrierEventClockMs + 1;

// Explicit compatibility escape hatch for PressureControlGUI. It is accepted
// only after the batch owner is already fail-stopped; a live production run can
// never be stolen. The legacy GUI applies its normal SAFE_STOP_VALUES next.
IF GuiReorientationLegacyTakeover AND ReorientationSafeLatch THEN
	GuiConveyorEnabled := FALSE;
	GuiArrayEnabled1 := FALSE;
	GuiArrayEnabled2 := FALSE;
	GuiArrayEnabled3 := FALSE;
	GuiArrayEnabled4 := FALSE;
	GuiReorientationControlActive := FALSE;
	GuiReorientationAbort := FALSE;
	GuiReorientationStart := FALSE;
	GuiReorientationFinish := FALSE;
	ReorientationFaultCode := 0;
	ReorientationState := 0;
	ReorientationSafeLatch := FALSE;
	ReorientationHeartbeatAlive := FALSE;
	BatchJobCount[1] := 0; BatchJobCount[2] := 0; BatchJobCount[3] := 0; BatchJobCount[4] := 0;
	BatchActiveSequence[1] := 0; BatchActiveSequence[2] := 0;
	BatchActiveSequence[3] := 0; BatchActiveSequence[4] := 0;
	GuiReorientationLegacyTakeover := FALSE;
END_IF

// A communication loss must remain safe and must never fall back to legacy control.
IF GuiReorientationControlActive THEN
	IF GuiReorientationHeartbeat <> ReorientationLastHeartbeat THEN
		ReorientationLastHeartbeat := GuiReorientationHeartbeat;
		ReorientationHeartbeatAck := GuiReorientationHeartbeat;
		ReorientationHeartbeatAgeMs := 0;
		ReorientationHeartbeatAlive := TRUE;
	ELSIF ReorientationHeartbeatAgeMs < 16#FFFFFFFF THEN
		ReorientationHeartbeatAgeMs := ReorientationHeartbeatAgeMs + 1;
	END_IF
	IF ReorientationHeartbeatAgeMs > 2000 THEN
		ReorientationHeartbeatAlive := FALSE;
		ReorientationFaultCode := 91;
		ReorientationState := 91;
		ReorientationSafeLatch := TRUE;
	END_IF
ELSIF NOT ReorientationSafeLatch THEN
	ReorientationHeartbeatAlive := FALSE;
	ReorientationState := 0;
END_IF

IF GuiReorientationReset AND GuiReorientationControlActive THEN
	ReorientationFaultCode := 0;
	ReorientationSafeLatch := FALSE;
	ReorientationState := 10;
	ReorientationHeartbeatAgeMs := 0;
	ReorientationLastHeartbeat := GuiReorientationHeartbeat;
	ReorientationHeartbeatAck := GuiReorientationHeartbeat;
	ReorientationHeartbeatAlive := TRUE;
	ReorientationComplete := FALSE;
	ReorientationExitSeen := FALSE;
	ReorientationTriggeredArrayMask := 0;
	ReorientationQueueEnqueueAck := 0;
	ReorientationQueueEnteredCount := 0;
	ReorientationQueueCompletedCount := 0;
	ReorientationQueueBypassCount := 0;
	ReorientationSensorSequence1 := 0;
	ReorientationSensorSequence2 := 0;
	ReorientationSensorSequence3 := 0;
	ReorientationSensorSequence4 := 0;
	ReorientationSensorSequence5 := 0;
	ReorientationSensorSequence6 := 0;
	ReorientationSensorSequence7 := 0;
	ReorientationSensorSequence8 := 0;
	ReorientationResultAvailable := FALSE;
	ReorientationResultSequence := 0;
	ReorientationResultTriggeredMask := 0;
	ReorientationResultFaultCode := 0;
	ReorientationFaultDetail := 0;
	ReorientationFaultSensor := 0;
	ReorientationFaultExpectedSequence := 0;
	ReorientationFaultPreviousSequence := 0;
	ReorientationFaultQueueAck := 0;
	ReorientationFaultQueueSlotSequence := 0;
	ReorientationFaultBarrierStableMask := 0;
	ReorientationWarningCode := 0;
	ReorientationWarningSensor := 0;
	ReorientationWarningSequence := 0;
	ReorientationWarningPreviousSequence := 0;
	ReorientationWarningSkippedBarrierMask := 0;
	ReorientationWarningCounter := 0;
	BatchNextCompleteSequence := 1;
	BatchLastAcceptedCommit := 0;
	BatchAcceptedResultAck := 0;
	GuiReorientationQueueCommit := 0;
	GuiReorientationQueueSequence := 0;
	GuiReorientationResultAck := 0;
	FOR BatchLoopIndex := 1 TO 8 DO
		BatchNextSensorSequence[BatchLoopIndex] := 1;
		BatchSensorSequence[BatchLoopIndex] := 0;
		BatchSensorNeedsClear[BatchLoopIndex] := FALSE;
	END_FOR
	FOR BatchLoopIndex := 1 TO 4 DO
		BatchJobHead[BatchLoopIndex] := 0;
		BatchJobTail[BatchLoopIndex] := 0;
		BatchJobCount[BatchLoopIndex] := 0;
		BatchActiveSequence[BatchLoopIndex] := 0;
		PairedFirstBarrierLocked[BatchLoopIndex] := FALSE;
		PairedFirstBarrierLockStartMs[BatchLoopIndex] := 0;
		PairedSecondBarrierLocked[BatchLoopIndex] := FALSE;
		PairedSecondBarrierLockStartMs[BatchLoopIndex] := 0;
	END_FOR
	// Reset is a command pulse. The PLC consumes it once so the GUI does not
	// need a separate reset/ready handshake just to lower the bit again.
	GuiReorientationReset := FALSE;
END_IF

IF GuiReorientationAbort AND GuiReorientationControlActive THEN
	ReorientationFaultCode := 90;
	ReorientationState := 90;
	ReorientationSafeLatch := TRUE;
END_IF

IF GuiReorientationControlActive AND (ReorientationState >= 20) AND (ReorientationState <= 30)
	AND (StepperPosError OR (ErrorCode0 <> 0) OR (ErrorCode1 <> 0)) THEN
	ReorientationFaultCode := 94;
	ReorientationState := 94;
	ReorientationSafeLatch := TRUE;
END_IF

IF ReorientationSafeLatch THEN
	GuiConveyorEnabled := FALSE;
	GuiArrayEnabled1 := FALSE;
	GuiArrayEnabled2 := FALSE;
	GuiArrayEnabled3 := FALSE;
	GuiArrayEnabled4 := FALSE;
	Array1TriggerPending := FALSE;
	Array2TriggerPending := FALSE;
	Array3TriggerPending := FALSE;
	Array4TriggerPending := FALSE;
END_IF

IF GuiResetVelocityEstimates THEN
	LastVelocityTimeMs := 0;
	LastVelocityTime2Ms := 0;
	LastVelocityTime3Ms := 0;
	LastVelocityTime4Ms := 0;
	VelocityTimingActive := FALSE;
	VelocityTiming2Active := FALSE;
	VelocityTiming3Active := FALSE;
	VelocityTiming4Active := FALSE;
	VelocityMeasurementValid := FALSE;
	VelocityMeasurement2Valid := FALSE;
	VelocityMeasurement3Valid := FALSE;
	VelocityMeasurement4Valid := FALSE;
	EstimatedVelocityMmPerSec := 0.0;
	EstimatedVelocityMmPerSec1 := 0.0;
	EstimatedVelocityMmPerSec2 := 0.0;
	EstimatedVelocityMmPerSec3 := 0.0;
	EstimatedVelocityMmPerSec4 := 0.0;
	EstimatedOffsetDelayMs1 := 0.0;
	EstimatedOffsetDelayMs2 := 0.0;
	EstimatedOffsetDelayMs3 := 0.0;
	EstimatedOffsetDelayMs4 := 0.0;
	OffsetDelayCycles1 := 0;
	OffsetDelayCycles2 := 0;
	OffsetDelayCycles3 := 0;
	OffsetDelayCycles4 := 0;
	GuiResetVelocityEstimates := FALSE;
END_IF

VelocityTimer(IN := VelocityTimingActive, PT := T#30S);
VelocityTimer2(IN := VelocityTiming2Active, PT := T#30S);
VelocityTimer3(IN := VelocityTiming3Active, PT := T#30S);
VelocityTimer4(IN := VelocityTiming4Active, PT := T#30S);

// Feed each idle array from its private FIFO.  The copied GUI-compatible fields
// are not touched again until this pulse has completed, so the existing VTEM
// state machines operate on an immutable per-part snapshot.
IF GuiReorientationControlActive AND ((ReorientationState = 20) OR (ReorientationState = 30)) THEN
	IF (State = 2) AND (BatchActiveSequence[1] = 0) AND (BatchJobCount[1] > 0) THEN
		BatchActiveSequence[1] := BatchJobSequence[BatchJobHead[1], 1];
		GuiPressureMbar1 := BatchJobPressureMbar[BatchJobHead[1], 1];
		GuiDelayMs1 := INT_TO_UINT(BatchJobDelayCycles[BatchJobHead[1], 1]);
		GuiPulseDurationMs1 := INT_TO_UINT(BatchJobPulseCycles[BatchJobHead[1], 1]);
		GuiOffsetMm1 := 0.0;
		GuiForceResponseDelayMs1 := 0.0;
		GuiForceSingleNozzleResponseDelayMs1 := 0.0;
		GuiArrayEnabled1 := TRUE;
		GuiNozzleEnabled1 := (BatchJobNozzleMask[BatchJobHead[1], 1] AND BYTE#1) <> BYTE#0;
		GuiNozzleEnabled2 := (BatchJobNozzleMask[BatchJobHead[1], 1] AND BYTE#2) <> BYTE#0;
		GuiNozzleEnabled3 := (BatchJobNozzleMask[BatchJobHead[1], 1] AND BYTE#4) <> BYTE#0;
		GuiNozzleEnabled4 := (BatchJobNozzleMask[BatchJobHead[1], 1] AND BYTE#8) <> BYTE#0;
		GuiNozzleEnabled5 := (BatchJobNozzleMask[BatchJobHead[1], 1] AND BYTE#16) <> BYTE#0;
		GuiNozzleEnabled6 := (BatchJobNozzleMask[BatchJobHead[1], 1] AND BYTE#32) <> BYTE#0;
		BatchJobHead[1] := (BatchJobHead[1] + 1) MOD 16;
		BatchJobCount[1] := BatchJobCount[1] - 1;
		Array1TriggerPending := TRUE;
	END_IF
	IF (State2 = 2) AND (BatchActiveSequence[2] = 0) AND (BatchJobCount[2] > 0) THEN
		BatchActiveSequence[2] := BatchJobSequence[BatchJobHead[2], 2];
		GuiPressureMbar2 := BatchJobPressureMbar[BatchJobHead[2], 2];
		GuiDelayMs2 := INT_TO_UINT(BatchJobDelayCycles[BatchJobHead[2], 2]);
		GuiPulseDurationMs2 := INT_TO_UINT(BatchJobPulseCycles[BatchJobHead[2], 2]);
		GuiOffsetMm2 := 0.0;
		GuiForceResponseDelayMs2 := 0.0;
		GuiForceSingleNozzleResponseDelayMs2 := 0.0;
		GuiArrayEnabled2 := TRUE;
		GuiNozzleEnabled7 := (BatchJobNozzleMask[BatchJobHead[2], 2] AND BYTE#1) <> BYTE#0;
		GuiNozzleEnabled8 := (BatchJobNozzleMask[BatchJobHead[2], 2] AND BYTE#2) <> BYTE#0;
		GuiNozzleEnabled9 := (BatchJobNozzleMask[BatchJobHead[2], 2] AND BYTE#4) <> BYTE#0;
		GuiNozzleEnabled10 := (BatchJobNozzleMask[BatchJobHead[2], 2] AND BYTE#8) <> BYTE#0;
		GuiNozzleEnabled11 := (BatchJobNozzleMask[BatchJobHead[2], 2] AND BYTE#16) <> BYTE#0;
		GuiNozzleEnabled12 := (BatchJobNozzleMask[BatchJobHead[2], 2] AND BYTE#32) <> BYTE#0;
		BatchJobHead[2] := (BatchJobHead[2] + 1) MOD 16;
		BatchJobCount[2] := BatchJobCount[2] - 1;
		Array2TriggerPending := TRUE;
	END_IF
	IF (State3 = 2) AND (BatchActiveSequence[3] = 0) AND (BatchJobCount[3] > 0) THEN
		BatchActiveSequence[3] := BatchJobSequence[BatchJobHead[3], 3];
		GuiPressureMbar3 := BatchJobPressureMbar[BatchJobHead[3], 3];
		GuiDelayMs3 := INT_TO_UINT(BatchJobDelayCycles[BatchJobHead[3], 3]);
		GuiPulseDurationMs3 := INT_TO_UINT(BatchJobPulseCycles[BatchJobHead[3], 3]);
		GuiOffsetMm3 := 0.0;
		GuiForceResponseDelayMs3 := 0.0;
		GuiForceSingleNozzleResponseDelayMs3 := 0.0;
		GuiArrayEnabled3 := TRUE;
		GuiNozzleEnabled13 := (BatchJobNozzleMask[BatchJobHead[3], 3] AND BYTE#1) <> BYTE#0;
		GuiNozzleEnabled14 := (BatchJobNozzleMask[BatchJobHead[3], 3] AND BYTE#2) <> BYTE#0;
		GuiNozzleEnabled15 := (BatchJobNozzleMask[BatchJobHead[3], 3] AND BYTE#4) <> BYTE#0;
		GuiNozzleEnabled16 := (BatchJobNozzleMask[BatchJobHead[3], 3] AND BYTE#8) <> BYTE#0;
		GuiNozzleEnabled17 := (BatchJobNozzleMask[BatchJobHead[3], 3] AND BYTE#16) <> BYTE#0;
		GuiNozzleEnabled18 := (BatchJobNozzleMask[BatchJobHead[3], 3] AND BYTE#32) <> BYTE#0;
		BatchJobHead[3] := (BatchJobHead[3] + 1) MOD 16;
		BatchJobCount[3] := BatchJobCount[3] - 1;
		Array3TriggerPending := TRUE;
	END_IF
	IF (State4 = 2) AND (BatchActiveSequence[4] = 0) AND (BatchJobCount[4] > 0) THEN
		BatchActiveSequence[4] := BatchJobSequence[BatchJobHead[4], 4];
		GuiPressureMbar4 := BatchJobPressureMbar[BatchJobHead[4], 4];
		GuiDelayMs4 := INT_TO_UINT(BatchJobDelayCycles[BatchJobHead[4], 4]);
		GuiPulseDurationMs4 := INT_TO_UINT(BatchJobPulseCycles[BatchJobHead[4], 4]);
		GuiOffsetMm4 := 0.0;
		GuiForceResponseDelayMs4 := 0.0;
		GuiForceSingleNozzleResponseDelayMs4 := 0.0;
		GuiArrayEnabled4 := TRUE;
		GuiNozzleEnabled19 := (BatchJobNozzleMask[BatchJobHead[4], 4] AND BYTE#1) <> BYTE#0;
		GuiNozzleEnabled20 := (BatchJobNozzleMask[BatchJobHead[4], 4] AND BYTE#2) <> BYTE#0;
		GuiNozzleEnabled21 := (BatchJobNozzleMask[BatchJobHead[4], 4] AND BYTE#4) <> BYTE#0;
		GuiNozzleEnabled22 := (BatchJobNozzleMask[BatchJobHead[4], 4] AND BYTE#8) <> BYTE#0;
		GuiNozzleEnabled23 := (BatchJobNozzleMask[BatchJobHead[4], 4] AND BYTE#16) <> BYTE#0;
		GuiNozzleEnabled24 := (BatchJobNozzleMask[BatchJobHead[4], 4] AND BYTE#32) <> BYTE#0;
		BatchJobHead[4] := (BatchJobHead[4] + 1) MOD 16;
		BatchJobCount[4] := BatchJobCount[4] - 1;
		Array4TriggerPending := TRUE;
	END_IF
END_IF

Array1Active := NOT GuiConveyorCalibrationMode AND NOT GuiVelocityCheckMode AND GuiArrayEnabled1 AND (GuiNozzleEnabled1 OR GuiNozzleEnabled2 OR GuiNozzleEnabled3 OR GuiNozzleEnabled4 OR GuiNozzleEnabled5 OR GuiNozzleEnabled6);
Array2Active := NOT GuiConveyorCalibrationMode AND NOT GuiVelocityCheckMode AND GuiArrayEnabled2 AND (GuiNozzleEnabled7 OR GuiNozzleEnabled8 OR GuiNozzleEnabled9 OR GuiNozzleEnabled10 OR GuiNozzleEnabled11 OR GuiNozzleEnabled12);
Array3Active := NOT GuiConveyorCalibrationMode AND NOT GuiVelocityCheckMode AND GuiArrayEnabled3 AND (GuiNozzleEnabled13 OR GuiNozzleEnabled14 OR GuiNozzleEnabled15 OR GuiNozzleEnabled16 OR GuiNozzleEnabled17 OR GuiNozzleEnabled18);
Array4Active := NOT GuiConveyorCalibrationMode AND NOT GuiVelocityCheckMode AND GuiArrayEnabled4 AND (GuiNozzleEnabled19 OR GuiNozzleEnabled20 OR GuiNozzleEnabled21 OR GuiNozzleEnabled22 OR GuiNozzleEnabled23 OR GuiNozzleEnabled24);

IF GuiConveyorSpeedMmPerSec < 0.0 THEN
	GuiConveyorSpeedMmPerSec := 0.0;
ELSIF GuiConveyorSpeedMmPerSec > 5000.0 THEN
	GuiConveyorSpeedMmPerSec := 5000.0;
END_IF

IF GuiConveyorMaxSpeedMmPerSec < 1.0 THEN
	GuiConveyorMaxSpeedMmPerSec := 1.0;
ELSIF GuiConveyorMaxSpeedMmPerSec > 5000.0 THEN
	GuiConveyorMaxSpeedMmPerSec := 5000.0;
END_IF

ConveyorSpeedMmPerSec := GuiConveyorSpeedMmPerSec;
IF ConveyorSpeedMmPerSec > GuiConveyorMaxSpeedMmPerSec THEN
	ConveyorSpeedMmPerSec := GuiConveyorMaxSpeedMmPerSec;
END_IF

IF GuiCalibrationMarkerDistanceMm < 1.0 THEN
	GuiCalibrationMarkerDistanceMm := 1.0;
ELSIF GuiCalibrationMarkerDistanceMm > 5000.0 THEN
	GuiCalibrationMarkerDistanceMm := 5000.0;
END_IF

IF GuiCalibrationJogSteps < 1 THEN
	GuiCalibrationJogSteps := 1;
ELSIF GuiCalibrationJogSteps > 100000 THEN
	GuiCalibrationJogSteps := 100000;
END_IF

IF GuiCalibrationJogSpeedFullStepsPerSec < 1.0 THEN
	GuiCalibrationJogSpeedFullStepsPerSec := 1.0;
ELSIF GuiCalibrationJogSpeedFullStepsPerSec > 500.0 THEN
	GuiCalibrationJogSpeedFullStepsPerSec := 500.0;
END_IF

// Entering calibration is fail-safe: normal belt motion remains disabled until explicitly re-enabled.
IF GuiConveyorCalibrationMode AND NOT LastConveyorCalibrationMode THEN
	GuiConveyorEnabled := FALSE;
	CalibrationLeftMarkValid := FALSE;
	CalibrationRightMarkValid := FALSE;
	CalibrationPositionDifferenceIncrements := 0;
	CalibrationFullStepDifference := 0.0;
	CalibrationStatusCode := 0;
END_IF
LastConveyorCalibrationMode := GuiConveyorCalibrationMode;

IF GuiBarrierCalibrationDebounceMs < 1 THEN
	GuiBarrierCalibrationDebounceMs := 1;
ELSIF GuiBarrierCalibrationDebounceMs > 200 THEN
	GuiBarrierCalibrationDebounceMs := 200;
END_IF

// All production timing and valve triggers use these shared, stable sensor states.
// Normalize the electrical polarity first. TRUE means clear beam and FALSE means part present.
LightBarrierLogical1 := LightBarrierOn1 <> GuiLightBarrierInvert1;
LightBarrierLogical2 := LightBarrierOn2 <> GuiLightBarrierInvert2;
LightBarrierLogical3 := LightBarrierOn3 <> GuiLightBarrierInvert3;
LightBarrierLogical4 := LightBarrierOn4 <> GuiLightBarrierInvert4;
LightBarrierLogical5 := LightBarrierOn5 <> GuiLightBarrierInvert5;
LightBarrierLogical6 := LightBarrierOn6 <> GuiLightBarrierInvert6;
LightBarrierLogical7 := LightBarrierOn7 <> GuiLightBarrierInvert7;
LightBarrierLogical8 := LightBarrierOn8 <> GuiLightBarrierInvert8;

// Changing polarity re-synchronizes the debouncer without generating an artificial edge.
IF (GuiLightBarrierInvert1 <> LastLightBarrierInvert1)
	OR (GuiLightBarrierInvert2 <> LastLightBarrierInvert2)
	OR (GuiLightBarrierInvert3 <> LastLightBarrierInvert3)
	OR (GuiLightBarrierInvert4 <> LastLightBarrierInvert4)
	OR (GuiLightBarrierInvert5 <> LastLightBarrierInvert5)
	OR (GuiLightBarrierInvert6 <> LastLightBarrierInvert6)
	OR (GuiLightBarrierInvert7 <> LastLightBarrierInvert7)
	OR (GuiLightBarrierInvert8 <> LastLightBarrierInvert8)
	OR (GuiLightBarrierDebounceEnabled1 <> LastLightBarrierDebounceEnabled1)
	OR (GuiLightBarrierDebounceEnabled2 <> LastLightBarrierDebounceEnabled2)
	OR (GuiLightBarrierDebounceEnabled3 <> LastLightBarrierDebounceEnabled3)
	OR (GuiLightBarrierDebounceEnabled4 <> LastLightBarrierDebounceEnabled4)
	OR (GuiLightBarrierDebounceEnabled5 <> LastLightBarrierDebounceEnabled5)
	OR (GuiLightBarrierDebounceEnabled6 <> LastLightBarrierDebounceEnabled6)
	OR (GuiLightBarrierDebounceEnabled7 <> LastLightBarrierDebounceEnabled7)
	OR (GuiLightBarrierDebounceEnabled8 <> LastLightBarrierDebounceEnabled8) THEN
	LightBarrierDebounceInitialized := FALSE;
	LightBarrierStableCounter1 := 0;
	LightBarrierStableCounter2 := 0;
	LightBarrierStableCounter3 := 0;
	LightBarrierStableCounter4 := 0;
	LightBarrierStableCounter5 := 0;
	LightBarrierStableCounter6 := 0;
	LightBarrierStableCounter7 := 0;
	LightBarrierStableCounter8 := 0;
END_IF
LastLightBarrierInvert1 := GuiLightBarrierInvert1;
LastLightBarrierInvert2 := GuiLightBarrierInvert2;
LastLightBarrierInvert3 := GuiLightBarrierInvert3;
LastLightBarrierInvert4 := GuiLightBarrierInvert4;
LastLightBarrierInvert5 := GuiLightBarrierInvert5;
LastLightBarrierInvert6 := GuiLightBarrierInvert6;
LastLightBarrierInvert7 := GuiLightBarrierInvert7;
LastLightBarrierInvert8 := GuiLightBarrierInvert8;
LastLightBarrierDebounceEnabled1 := GuiLightBarrierDebounceEnabled1;
LastLightBarrierDebounceEnabled2 := GuiLightBarrierDebounceEnabled2;
LastLightBarrierDebounceEnabled3 := GuiLightBarrierDebounceEnabled3;
LastLightBarrierDebounceEnabled4 := GuiLightBarrierDebounceEnabled4;
LastLightBarrierDebounceEnabled5 := GuiLightBarrierDebounceEnabled5;
LastLightBarrierDebounceEnabled6 := GuiLightBarrierDebounceEnabled6;
LastLightBarrierDebounceEnabled7 := GuiLightBarrierDebounceEnabled7;
LastLightBarrierDebounceEnabled8 := GuiLightBarrierDebounceEnabled8;

// On startup, synchronize without creating a false edge.
IF NOT LightBarrierDebounceInitialized THEN
	LightBarrierStable1 := LightBarrierLogical1;
	LightBarrierStable2 := LightBarrierLogical2;
	LightBarrierStable3 := LightBarrierLogical3;
	LightBarrierStable4 := LightBarrierLogical4;
	LightBarrierStable5 := LightBarrierLogical5;
	LightBarrierStable6 := LightBarrierLogical6;
	LightBarrierStable7 := LightBarrierLogical7;
	LightBarrierStable8 := LightBarrierLogical8;
	LastLightBarrier1 := LightBarrierLogical1;
	LastLightBarrier2 := LightBarrierLogical2;
	LastLightBarrier3 := LightBarrierLogical3;
	LastLightBarrier4 := LightBarrierLogical4;
	LastLightBarrier5 := LightBarrierLogical5;
	LastLightBarrier6 := LightBarrierLogical6;
	LastLightBarrier7 := LightBarrierLogical7;
	LastLightBarrier8 := LightBarrierLogical8;
	LightBarrierStableCounter1 := 0;
	LightBarrierStableCounter2 := 0;
	LightBarrierStableCounter3 := 0;
	LightBarrierStableCounter4 := 0;
	LightBarrierStableCounter5 := 0;
	LightBarrierStableCounter6 := 0;
	LightBarrierStableCounter7 := 0;
	LightBarrierStableCounter8 := 0;
	LightBarrierDebounceInitialized := TRUE;
ELSE
	IF NOT GuiLightBarrierDebounceEnabled1 THEN
		LightBarrierStable1 := LightBarrierLogical1;
		LightBarrierStableCounter1 := 0;
	ELSIF LightBarrierLogical1 <> LightBarrierStable1 THEN
		IF LightBarrierStableCounter1 < GuiBarrierCalibrationDebounceMs THEN
			LightBarrierStableCounter1 := LightBarrierStableCounter1 + 1;
		END_IF
		IF LightBarrierStableCounter1 >= GuiBarrierCalibrationDebounceMs THEN
			LightBarrierStable1 := LightBarrierLogical1;
			LightBarrierStableCounter1 := 0;
		END_IF
	ELSE
		LightBarrierStableCounter1 := 0;
	END_IF
	IF NOT GuiLightBarrierDebounceEnabled2 THEN
		LightBarrierStable2 := LightBarrierLogical2;
		LightBarrierStableCounter2 := 0;
	ELSIF LightBarrierLogical2 <> LightBarrierStable2 THEN
		IF LightBarrierStableCounter2 < GuiBarrierCalibrationDebounceMs THEN
			LightBarrierStableCounter2 := LightBarrierStableCounter2 + 1;
		END_IF
		IF LightBarrierStableCounter2 >= GuiBarrierCalibrationDebounceMs THEN
			LightBarrierStable2 := LightBarrierLogical2;
			LightBarrierStableCounter2 := 0;
		END_IF
	ELSE
		LightBarrierStableCounter2 := 0;
	END_IF
	IF NOT GuiLightBarrierDebounceEnabled3 THEN
		LightBarrierStable3 := LightBarrierLogical3;
		LightBarrierStableCounter3 := 0;
	ELSIF LightBarrierLogical3 <> LightBarrierStable3 THEN
		IF LightBarrierStableCounter3 < GuiBarrierCalibrationDebounceMs THEN
			LightBarrierStableCounter3 := LightBarrierStableCounter3 + 1;
		END_IF
		IF LightBarrierStableCounter3 >= GuiBarrierCalibrationDebounceMs THEN
			LightBarrierStable3 := LightBarrierLogical3;
			LightBarrierStableCounter3 := 0;
		END_IF
	ELSE
		LightBarrierStableCounter3 := 0;
	END_IF
	IF NOT GuiLightBarrierDebounceEnabled4 THEN
		LightBarrierStable4 := LightBarrierLogical4;
		LightBarrierStableCounter4 := 0;
	ELSIF LightBarrierLogical4 <> LightBarrierStable4 THEN
		IF LightBarrierStableCounter4 < GuiBarrierCalibrationDebounceMs THEN
			LightBarrierStableCounter4 := LightBarrierStableCounter4 + 1;
		END_IF
		IF LightBarrierStableCounter4 >= GuiBarrierCalibrationDebounceMs THEN
			LightBarrierStable4 := LightBarrierLogical4;
			LightBarrierStableCounter4 := 0;
		END_IF
	ELSE
		LightBarrierStableCounter4 := 0;
	END_IF
	IF NOT GuiLightBarrierDebounceEnabled5 THEN
		LightBarrierStable5 := LightBarrierLogical5;
		LightBarrierStableCounter5 := 0;
	ELSIF LightBarrierLogical5 <> LightBarrierStable5 THEN
		IF LightBarrierStableCounter5 < GuiBarrierCalibrationDebounceMs THEN
			LightBarrierStableCounter5 := LightBarrierStableCounter5 + 1;
		END_IF
		IF LightBarrierStableCounter5 >= GuiBarrierCalibrationDebounceMs THEN
			LightBarrierStable5 := LightBarrierLogical5;
			LightBarrierStableCounter5 := 0;
		END_IF
	ELSE
		LightBarrierStableCounter5 := 0;
	END_IF
	IF NOT GuiLightBarrierDebounceEnabled6 THEN
		LightBarrierStable6 := LightBarrierLogical6;
		LightBarrierStableCounter6 := 0;
	ELSIF LightBarrierLogical6 <> LightBarrierStable6 THEN
		IF LightBarrierStableCounter6 < GuiBarrierCalibrationDebounceMs THEN
			LightBarrierStableCounter6 := LightBarrierStableCounter6 + 1;
		END_IF
		IF LightBarrierStableCounter6 >= GuiBarrierCalibrationDebounceMs THEN
			LightBarrierStable6 := LightBarrierLogical6;
			LightBarrierStableCounter6 := 0;
		END_IF
	ELSE
		LightBarrierStableCounter6 := 0;
	END_IF
	IF NOT GuiLightBarrierDebounceEnabled7 THEN
		LightBarrierStable7 := LightBarrierLogical7;
		LightBarrierStableCounter7 := 0;
	ELSIF LightBarrierLogical7 <> LightBarrierStable7 THEN
		IF LightBarrierStableCounter7 < GuiBarrierCalibrationDebounceMs THEN
			LightBarrierStableCounter7 := LightBarrierStableCounter7 + 1;
		END_IF
		IF LightBarrierStableCounter7 >= GuiBarrierCalibrationDebounceMs THEN
			LightBarrierStable7 := LightBarrierLogical7;
			LightBarrierStableCounter7 := 0;
		END_IF
	ELSE
		LightBarrierStableCounter7 := 0;
	END_IF
	IF NOT GuiLightBarrierDebounceEnabled8 THEN
		LightBarrierStable8 := LightBarrierLogical8;
		LightBarrierStableCounter8 := 0;
	ELSIF LightBarrierLogical8 <> LightBarrierStable8 THEN
		IF LightBarrierStableCounter8 < GuiBarrierCalibrationDebounceMs THEN
			LightBarrierStableCounter8 := LightBarrierStableCounter8 + 1;
		END_IF
		IF LightBarrierStableCounter8 >= GuiBarrierCalibrationDebounceMs THEN
			LightBarrierStable8 := LightBarrierLogical8;
			LightBarrierStableCounter8 := 0;
		END_IF
	ELSE
		LightBarrierStableCounter8 := 0;
	END_IF
END_IF

CASE GuiBarrierCalibrationFirstSensor OF
	1: BarrierCalibrationFirstState := LightBarrierLogical1;
	2: BarrierCalibrationFirstState := LightBarrierLogical2;
	3: BarrierCalibrationFirstState := LightBarrierLogical3;
	4: BarrierCalibrationFirstState := LightBarrierLogical4;
	5: BarrierCalibrationFirstState := LightBarrierLogical5;
	6: BarrierCalibrationFirstState := LightBarrierLogical6;
	7: BarrierCalibrationFirstState := LightBarrierLogical7;
	8: BarrierCalibrationFirstState := LightBarrierLogical8;
ELSE
	BarrierCalibrationFirstState := FALSE;
END_CASE

CASE GuiBarrierCalibrationSecondSensor OF
	1: BarrierCalibrationSecondState := LightBarrierLogical1;
	2: BarrierCalibrationSecondState := LightBarrierLogical2;
	3: BarrierCalibrationSecondState := LightBarrierLogical3;
	4: BarrierCalibrationSecondState := LightBarrierLogical4;
	5: BarrierCalibrationSecondState := LightBarrierLogical5;
	6: BarrierCalibrationSecondState := LightBarrierLogical6;
	7: BarrierCalibrationSecondState := LightBarrierLogical7;
	8: BarrierCalibrationSecondState := LightBarrierLogical8;
ELSE
	BarrierCalibrationSecondState := FALSE;
END_CASE

// Prepare a light-barrier spacing measurement before the GUI starts a long relative move.
IF GuiBarrierCalibrationStart THEN
	IF GuiConveyorCalibrationMode
		AND GuiConveyorCalibrationValid
		AND (GuiConveyorMmPerFullStep > 0.0)
		AND (ConveyorMotionState = 0)
		AND NOT StepperPosBusy
		AND StepperPosReadyToExecute
		AND (GuiBarrierCalibrationFirstSensor >= 1)
		AND (GuiBarrierCalibrationFirstSensor <= 8)
		AND (GuiBarrierCalibrationSecondSensor >= 1)
		AND (GuiBarrierCalibrationSecondSensor <= 8)
		AND (GuiBarrierCalibrationFirstSensor <> GuiBarrierCalibrationSecondSensor) THEN
		BarrierCalibrationActive := TRUE;
		BarrierCalibrationFirstCaptured := FALSE;
		BarrierCalibrationSecondCaptured := FALSE;
		BarrierCalibrationValid := FALSE;
		BarrierCalibrationFirstPosition := 0;
		BarrierCalibrationSecondPosition := 0;
		BarrierCalibrationDifferenceIncrements := 0;
		BarrierCalibrationDistanceMm := 0.0;
		BarrierCalibrationFirstInitialState := BarrierCalibrationFirstState;
		BarrierCalibrationSecondInitialState := BarrierCalibrationSecondState;
		BarrierCalibrationFirstCandidatePosition := 0;
		BarrierCalibrationSecondCandidatePosition := 0;
		BarrierCalibrationFirstStableCycles := 0;
		BarrierCalibrationSecondStableCycles := 0;
		BarrierCalibrationStatusCode := 1;
	ELSE
		BarrierCalibrationActive := FALSE;
		BarrierCalibrationStatusCode := 4;
		GuiCalibrationMoveRight := FALSE;
	END_IF
	GuiBarrierCalibrationStart := FALSE;
END_IF

IF GuiConveyorCalibrationValid AND (GuiConveyorMmPerFullStep > 0.0) THEN
	CalibrationStepsPerMm := 1.0 / GuiConveyorMmPerFullStep;
ELSE
	GuiConveyorCalibrationValid := FALSE;
	CalibrationStepsPerMm := 0.0;
END_IF

// Capture either marker only while the terminal is stationary.
IF GuiCalibrationCaptureLeftMark THEN
	IF GuiConveyorCalibrationMode AND (ConveyorMotionState = 0) AND NOT StepperPosBusy
		AND StepperPosReadyToExecute AND NOT StepperPosError THEN
		CalibrationLeftPosition := StepperInternalPosition;
		CalibrationLeftMarkValid := TRUE;
		CalibrationStatusCode := 0;
	ELSE
		CalibrationStatusCode := 4;
	END_IF
	GuiCalibrationCaptureLeftMark := FALSE;
END_IF

IF GuiCalibrationCaptureRightMark THEN
	IF GuiConveyorCalibrationMode AND (ConveyorMotionState = 0) AND NOT StepperPosBusy
		AND StepperPosReadyToExecute AND NOT StepperPosError THEN
		CalibrationRightPosition := StepperInternalPosition;
		CalibrationRightMarkValid := TRUE;
		CalibrationStatusCode := 0;
	ELSE
		CalibrationStatusCode := 4;
	END_IF
	GuiCalibrationCaptureRightMark := FALSE;
END_IF

// Recalculate whenever both positions or the physical marker spacing change.
IF GuiConveyorCalibrationMode AND CalibrationLeftMarkValid AND CalibrationRightMarkValid THEN
	// Modular counter difference works across both the sign boundary and UDINT wrap.
	CalibrationPositionDelta := UDINT_TO_LINT(CalibrationRightPosition)
		- UDINT_TO_LINT(CalibrationLeftPosition);
	IF CalibrationPositionDelta > LINT#2147483647 THEN
		CalibrationPositionDelta := CalibrationPositionDelta - LINT#4294967296;
	ELSIF CalibrationPositionDelta < LINT#-2147483648 THEN
		CalibrationPositionDelta := CalibrationPositionDelta + LINT#4294967296;
	END_IF
	IF CalibrationPositionDelta < 0 THEN
		CalibrationPositionDelta := -CalibrationPositionDelta;
	END_IF
	IF CalibrationPositionDelta > 0 THEN
		CalibrationPositionDifferenceIncrements := LINT_TO_UDINT(CalibrationPositionDelta);
		CalibrationFullStepDifference := TO_REAL(CalibrationPositionDifferenceIncrements) / 64.0;
		GuiConveyorMmPerFullStep := GuiCalibrationMarkerDistanceMm / CalibrationFullStepDifference;
		ConveyorServoCalibratedMmPerFullStep := GuiConveyorMmPerFullStep;
		CalibrationStepsPerMm := 1.0 / GuiConveyorMmPerFullStep;
		GuiConveyorCalibrationValid := TRUE;
	ELSE
		CalibrationPositionDifferenceIncrements := 0;
		CalibrationFullStepDifference := 0.0;
		CalibrationStatusCode := 4;
	END_IF
END_IF

// Convert the physical speed request to the 0..10000 positioning-interface velocity range.
IF GuiConveyorCalibrationValid AND (GuiConveyorMmPerFullStep > 0.0) THEN
	ConveyorFullStepsPerSec := ConveyorSpeedMmPerSec / GuiConveyorMmPerFullStep;
	ConveyorVelocityRatio := ConveyorFullStepsPerSec / ConveyorSpeedRangeFullStepsPerSec;
ELSE
	ConveyorFullStepsPerSec := 0.0;
	ConveyorVelocityRatio := 0.0;
END_IF
IF ConveyorVelocityRatio < 0.0 THEN
	ConveyorVelocityRatio := 0.0;
ELSIF ConveyorVelocityRatio > 1.0 THEN
	ConveyorVelocityRatio := 1.0;
END_IF
ConveyorVelocityRaw := REAL_TO_INT(ConveyorVelocityRatio * 10000.0);

// A calibration move is a finite relative positioning command in motor full steps.
IF GuiCalibrationMoveLeft OR GuiCalibrationMoveRight THEN
	IF GuiConveyorCalibrationMode
		AND (ConveyorMotionState = 0)
		AND NOT StepperPosBusy
		AND StepperPosReadyToExecute
		AND (GuiCalibrationMoveLeft <> GuiCalibrationMoveRight) THEN
		CalibrationTargetIncrements := UDINT_TO_DINT(GuiCalibrationJogSteps * UDINT#64);
		CalibrationDirectionNegative := GuiCalibrationMoveLeft;
		IF GuiConveyorReverse THEN
			CalibrationDirectionNegative := NOT CalibrationDirectionNegative;
		END_IF
		IF CalibrationDirectionNegative THEN
			CalibrationTargetIncrements := -CalibrationTargetIncrements;
		END_IF
		ConveyorActiveVelocity := REAL_TO_INT(
			GuiCalibrationJogSpeedFullStepsPerSec / ConveyorSpeedRangeFullStepsPerSec * 10000.0);
		IF ConveyorActiveVelocity < 1 THEN
			ConveyorActiveVelocity := 1;
		ELSIF ConveyorActiveVelocity > 10000 THEN
			ConveyorActiveVelocity := 10000;
		END_IF
		ConveyorActiveStartType := 2; //RELATIVE
		// Keep the cyclic command words at zero until the positioning interface reports ready.
		StepperPosTargetPosition := 0;
		StepperPosVelocity := 0;
		StepperPosStartType := 0;
		ConveyorMotionMode := 2;
		ConveyorMotionState := 10;
		CalibrationStatusCode := 1;
	ELSE
		CalibrationStatusCode := 4;
	END_IF
	GuiCalibrationMoveLeft := FALSE;
	GuiCalibrationMoveRight := FALSE;
END_IF

// One state machine owns all positioning-interface commands.
CASE ConveyorMotionState OF
	0:
		StepperPosExecute := FALSE;
		StepperPosEmergencyStop := FALSE;
		StepperPosTargetPosition := 0;
		StepperPosVelocity := 0;
		StepperPosStartType := 0;
		StepperPosAcceleration := 1000;
		StepperPosDeceleration := 1000;
		ConveyorMotionMode := 0;
		IF GuiConveyorEnabled AND NOT GuiConveyorCalibrationMode AND (ConveyorVelocityRaw > 0) THEN
			IF GuiConveyorReverse THEN
				ConveyorActiveStartType := 4; //ENDLESS_MINUS
			ELSE
				ConveyorActiveStartType := 3; //ENDLESS_PLUS
			END_IF
			ConveyorActiveVelocity := ConveyorVelocityRaw;
			ConveyorMotionMode := 1;
			ConveyorMotionState := 10;
		END_IF

	10:
		StepperPosExecute := FALSE;
		IF StepperPosError THEN
			ConveyorMotionState := 50;
			CalibrationStatusCode := 5;
		ELSIF GuiCalibrationStop
			OR ((ConveyorMotionMode = 2) AND NOT GuiConveyorCalibrationMode)
			OR ((ConveyorMotionMode = 1) AND ((NOT GuiConveyorEnabled) OR GuiConveyorCalibrationMode)) THEN
			StepperPosEmergencyStop := TRUE;
			ConveyorMotionState := 40;
		ELSIF StepperPosReadyToExecute THEN
			IF ConveyorMotionMode = 2 THEN
				StepperPosTargetPosition := DINT_TO_UDINT(CalibrationTargetIncrements);
			ELSE
				StepperPosTargetPosition := 0;
			END_IF
			StepperPosVelocity := ConveyorActiveVelocity;
			StepperPosStartType := ConveyorActiveStartType;
			StepperPosAcceleration := 1000;
			StepperPosDeceleration := 1000;
			StepperPosExecute := TRUE;
			ConveyorMotionState := 20;
		END_IF

	20:
		StepperPosExecute := TRUE;
		IF StepperPosError THEN
			StepperPosExecute := FALSE;
			ConveyorMotionState := 50;
			CalibrationStatusCode := 5;
		ELSIF GuiCalibrationStop
			OR ((ConveyorMotionMode = 2) AND NOT GuiConveyorCalibrationMode)
			OR ((ConveyorMotionMode = 1) AND ((NOT GuiConveyorEnabled) OR GuiConveyorCalibrationMode)) THEN
			StepperPosEmergencyStop := TRUE;
			StepperPosExecute := FALSE;
			ConveyorMotionState := 40;
		ELSIF StepperPosBusy THEN
			ConveyorMotionState := 30;
			IF ConveyorMotionMode = 2 THEN
				CalibrationStatusCode := 2;
			END_IF
		END_IF

	30:
		StepperPosExecute := TRUE;
		IF StepperPosError THEN
			StepperPosExecute := FALSE;
			ConveyorMotionState := 50;
			CalibrationStatusCode := 5;
		ELSIF GuiCalibrationStop OR ((ConveyorMotionMode = 2) AND NOT GuiConveyorCalibrationMode) THEN
			StepperPosEmergencyStop := TRUE;
			StepperPosExecute := FALSE;
			ConveyorMotionState := 40;
		ELSIF ConveyorMotionMode = 2 THEN
			IF NOT StepperPosBusy THEN
				StepperPosExecute := FALSE;
				ConveyorMotionState := 0;
				ConveyorMotionMode := 0;
				CalibrationStatusCode := 3;
			END_IF
		ELSIF (NOT GuiConveyorEnabled)
			OR GuiConveyorCalibrationMode
			OR (ConveyorVelocityRaw <> ConveyorActiveVelocity)
			OR ((GuiConveyorReverse AND (ConveyorActiveStartType <> 4))
				OR ((NOT GuiConveyorReverse) AND (ConveyorActiveStartType <> 3))) THEN
			StepperPosExecute := FALSE;
			ConveyorMotionState := 40;
		ELSIF NOT StepperPosBusy THEN
			StepperPosExecute := FALSE;
			ConveyorMotionState := 0;
			ConveyorMotionMode := 0;
		END_IF

	40:
		StepperPosExecute := FALSE;
		IF NOT StepperPosBusy THEN
			StepperPosEmergencyStop := FALSE;
			ConveyorMotionState := 0;
			ConveyorMotionMode := 0;
		END_IF

	50:
		StepperPosExecute := FALSE;
		StepperPosEmergencyStop := FALSE;
		IF NOT StepperPosError THEN
			ConveyorMotionState := 0;
			ConveyorMotionMode := 0;
		END_IF
ELSE
	ConveyorMotionState := 0;
	ConveyorMotionMode := 0;
	StepperPosExecute := FALSE;
	StepperPosEmergencyStop := FALSE;
END_CASE

CalibrationBusy := (ConveyorMotionMode = 2) AND (ConveyorMotionState <> 0);
CalibrationError := StepperPosError;
StepperControlEnable := GuiConveyorCalibrationMode OR GuiConveyorEnabled OR (ConveyorMotionState <> 0);
StepperControlReset := GuiConveyorReset;
GuiConveyorReset := FALSE;
StepperControlReduceTorque := StepperControlEnable AND (ConveyorMotionState = 0) AND NOT StepperPosBusy;
StepperControlDigitalOutput1 := FALSE;
BarrierCalibrationAbortRequested := GuiCalibrationStop
	OR NOT GuiConveyorCalibrationMode
	OR StepperPosError;
GuiCalibrationStop := FALSE;

LightBarrier1FallingEdge := (NOT LightBarrierStable1) AND LastLightBarrier1;
LightBarrier2FallingEdge := (NOT LightBarrierStable2) AND LastLightBarrier2;
LightBarrier3FallingEdge := (NOT LightBarrierStable3) AND LastLightBarrier3;
LightBarrier4FallingEdge := (NOT LightBarrierStable4) AND LastLightBarrier4;
LightBarrier5FallingEdge := (NOT LightBarrierStable5) AND LastLightBarrier5;
LightBarrier6FallingEdge := (NOT LightBarrierStable6) AND LastLightBarrier6;
LightBarrier7FallingEdge := (NOT LightBarrierStable7) AND LastLightBarrier7;
LightBarrier8FallingEdge := (NOT LightBarrierStable8) AND LastLightBarrier8;

// Alternating pair gate. A workpiece can expose more than one optical edge at
// either barrier. After the first barrier fires, only the second barrier can
// release it; after the second fires, only the next accepted first-barrier edge
// can release it. Both locks also expire after 500 ms. Raw/stable transitions
// above remain available unchanged for diagnostics and calibration.
FOR BatchLoopIndex := 1 TO 4 DO
	IF PairedFirstBarrierLocked[BatchLoopIndex]
		AND ((LightBarrierEventClockMs - PairedFirstBarrierLockStartMs[BatchLoopIndex])
			>= PairedBarrierLockTimeoutMs) THEN
		PairedFirstBarrierLocked[BatchLoopIndex] := FALSE;
	END_IF
	IF PairedSecondBarrierLocked[BatchLoopIndex]
		AND ((LightBarrierEventClockMs - PairedSecondBarrierLockStartMs[BatchLoopIndex])
			>= PairedBarrierLockTimeoutMs) THEN
		PairedSecondBarrierLocked[BatchLoopIndex] := FALSE;
	END_IF
END_FOR

// Evaluate the second barrier first. This lets a simultaneous second edge for
// the old workpiece release the first edge of the following workpiece.
PairedSecondBarrierFalling[1] := LightBarrier2FallingEdge AND NOT PairedSecondBarrierLocked[1];
PairedSecondBarrierFalling[2] := LightBarrier4FallingEdge AND NOT PairedSecondBarrierLocked[2];
PairedSecondBarrierFalling[3] := LightBarrier6FallingEdge AND NOT PairedSecondBarrierLocked[3];
PairedSecondBarrierFalling[4] := LightBarrier8FallingEdge AND NOT PairedSecondBarrierLocked[4];

FOR BatchLoopIndex := 1 TO 4 DO
	IF PairedSecondBarrierFalling[BatchLoopIndex] THEN
		PairedSecondBarrierLocked[BatchLoopIndex] := TRUE;
		PairedSecondBarrierLockStartMs[BatchLoopIndex] := LightBarrierEventClockMs;
		PairedFirstBarrierLocked[BatchLoopIndex] := FALSE;
	END_IF
END_FOR

PairedFirstBarrierFalling[1] := LightBarrier1FallingEdge AND NOT PairedFirstBarrierLocked[1];
PairedFirstBarrierFalling[2] := LightBarrier3FallingEdge AND NOT PairedFirstBarrierLocked[2];
PairedFirstBarrierFalling[3] := LightBarrier5FallingEdge AND NOT PairedFirstBarrierLocked[3];
PairedFirstBarrierFalling[4] := LightBarrier7FallingEdge AND NOT PairedFirstBarrierLocked[4];

FOR BatchLoopIndex := 1 TO 4 DO
	IF PairedFirstBarrierFalling[BatchLoopIndex] THEN
		PairedFirstBarrierLocked[BatchLoopIndex] := TRUE;
		PairedFirstBarrierLockStartMs[BatchLoopIndex] := LightBarrierEventClockMs;
		PairedSecondBarrierLocked[BatchLoopIndex] := FALSE;
	END_IF
END_FOR

// Capture the exact gate BOOLs, including their return to FALSE next cycle.
// This diagnostic buffer never participates in trigger or velocity decisions.
LightBarrierFilteredSignal[1] := PairedFirstBarrierFalling[1];
LightBarrierFilteredSignal[2] := PairedSecondBarrierFalling[1];
LightBarrierFilteredSignal[3] := PairedFirstBarrierFalling[2];
LightBarrierFilteredSignal[4] := PairedSecondBarrierFalling[2];
LightBarrierFilteredSignal[5] := PairedFirstBarrierFalling[3];
LightBarrierFilteredSignal[6] := PairedSecondBarrierFalling[3];
LightBarrierFilteredSignal[7] := PairedFirstBarrierFalling[4];
LightBarrierFilteredSignal[8] := PairedSecondBarrierFalling[4];
LightBarrierFilteredEventHistory[0] := 1;
LightBarrierFilteredEventHistory[2] := LightBarrierEventClockMs;
FOR LightBarrierFilteredSensor := 1 TO 8 DO
	IF LightBarrierFilteredSignal[LightBarrierFilteredSensor] <> LastLightBarrierFilteredSignal[LightBarrierFilteredSensor] THEN
		LightBarrierFilteredSlot := 3 + (((LightBarrierFilteredEventHistory[1] + 1) MOD 256) * 3);
		LightBarrierFilteredEventHistory[LightBarrierFilteredSlot + 1] := LightBarrierEventClockMs;
		LightBarrierFilteredEventHistory[LightBarrierFilteredSlot + 2] := INT_TO_UDINT(LightBarrierFilteredSensor) * 2
			+ BOOL_TO_UDINT(LightBarrierFilteredSignal[LightBarrierFilteredSensor]);
		LightBarrierFilteredEventHistory[LightBarrierFilteredSlot] := LightBarrierFilteredEventHistory[1] + 1;
		LightBarrierFilteredEventHistory[1] := LightBarrierFilteredEventHistory[LightBarrierFilteredSlot];
	END_IF
	LastLightBarrierFilteredSignal[LightBarrierFilteredSensor] := LightBarrierFilteredSignal[LightBarrierFilteredSensor];
END_FOR

// Production-run ownership.  State 20 accepts parts continuously; state 30
// refuses new commits and drains the already accepted queue.
IF GuiReorientationControlActive AND (ReorientationState = 0) THEN
	ReorientationState := 10;
END_IF
IF GuiReorientationControlActive AND GuiReorientationStart AND (ReorientationState = 10) AND ReorientationHeartbeatAlive AND NOT ReorientationSafeLatch THEN
	ReorientationExpectedArrayMask := 0;
	ReorientationTriggeredArrayMask := 0;
	ReorientationExitSeen := FALSE;
	ReorientationComplete := FALSE;
	ReorientationState := 20;
END_IF

IF GuiReorientationControlActive AND GuiReorientationFinish AND (ReorientationState = 20) THEN
	ReorientationState := 30;
END_IF

// Atomic producer commit.  Sequence IDs must be contiguous and an unacknowledged
// result keeps its ring slot occupied, preventing silent overwrite.
IF GuiReorientationControlActive AND (ReorientationState = 20)
	AND (GuiReorientationQueueCommit <> BatchLastAcceptedCommit) THEN
	IF (GuiReorientationQueueCommit <> (ReorientationQueueEnqueueAck + 1))
		OR (GuiReorientationQueueSequence <> GuiReorientationQueueCommit) THEN
		ReorientationFaultCode := 92;
		ReorientationState := 92;
		ReorientationSafeLatch := TRUE;
	ELSIF (ReorientationQueueEnqueueAck - BatchAcceptedResultAck) >= 128 THEN
		ReorientationFaultCode := 93;
		ReorientationState := 93;
		ReorientationSafeLatch := TRUE;
	ELSE
		BatchSlotIndex := UDINT_TO_INT((GuiReorientationQueueSequence - 1) MOD 128);
		BatchQueueSequence[BatchSlotIndex] := GuiReorientationQueueSequence;
		BatchQueueTrackId[BatchSlotIndex] := GuiReorientationQueueTrackId;
		BatchQueuePoseId[BatchSlotIndex] := GuiReorientationQueuePoseId;
		BatchQueueDecisionCode[BatchSlotIndex] := GuiReorientationQueueDecisionCode;
		BatchQueueArrayMask[BatchSlotIndex] := GuiReorientationQueueArrayMask AND BYTE#15;
		BatchQueueNozzleMask[BatchSlotIndex, 1] := GuiReorientationQueueNozzleMask1 AND BYTE#63;
		BatchQueueNozzleMask[BatchSlotIndex, 2] := GuiReorientationQueueNozzleMask2 AND BYTE#63;
		BatchQueueNozzleMask[BatchSlotIndex, 3] := GuiReorientationQueueNozzleMask3 AND BYTE#63;
		BatchQueueNozzleMask[BatchSlotIndex, 4] := GuiReorientationQueueNozzleMask4 AND BYTE#63;
		BatchQueuePressureMbar[BatchSlotIndex, 1] := GuiReorientationQueuePressureMbar1;
		BatchQueuePressureMbar[BatchSlotIndex, 2] := GuiReorientationQueuePressureMbar2;
		BatchQueuePressureMbar[BatchSlotIndex, 3] := GuiReorientationQueuePressureMbar3;
		BatchQueuePressureMbar[BatchSlotIndex, 4] := GuiReorientationQueuePressureMbar4;
		BatchQueueDelayMs[BatchSlotIndex, 1] := GuiReorientationQueueDelayMs1;
		BatchQueueDelayMs[BatchSlotIndex, 2] := GuiReorientationQueueDelayMs2;
		BatchQueueDelayMs[BatchSlotIndex, 3] := GuiReorientationQueueDelayMs3;
		BatchQueueDelayMs[BatchSlotIndex, 4] := GuiReorientationQueueDelayMs4;
		BatchQueuePulseMs[BatchSlotIndex, 1] := GuiReorientationQueuePulseMs1;
		BatchQueuePulseMs[BatchSlotIndex, 2] := GuiReorientationQueuePulseMs2;
		BatchQueuePulseMs[BatchSlotIndex, 3] := GuiReorientationQueuePulseMs3;
		BatchQueuePulseMs[BatchSlotIndex, 4] := GuiReorientationQueuePulseMs4;
		BatchQueueOffsetMm[BatchSlotIndex, 1] := GuiReorientationQueueOffsetMm1;
		BatchQueueOffsetMm[BatchSlotIndex, 2] := GuiReorientationQueueOffsetMm2;
		BatchQueueOffsetMm[BatchSlotIndex, 3] := GuiReorientationQueueOffsetMm3;
		BatchQueueOffsetMm[BatchSlotIndex, 4] := GuiReorientationQueueOffsetMm4;
		BatchQueueForceResponseMs[BatchSlotIndex, 1] := GuiReorientationQueueForceResponseMs1;
		BatchQueueForceResponseMs[BatchSlotIndex, 2] := GuiReorientationQueueForceResponseMs2;
		BatchQueueForceResponseMs[BatchSlotIndex, 3] := GuiReorientationQueueForceResponseMs3;
		BatchQueueForceResponseMs[BatchSlotIndex, 4] := GuiReorientationQueueForceResponseMs4;
		BatchQueueForceSingleMs[BatchSlotIndex, 1] := GuiReorientationQueueForceSingleMs1;
		BatchQueueForceSingleMs[BatchSlotIndex, 2] := GuiReorientationQueueForceSingleMs2;
		BatchQueueForceSingleMs[BatchSlotIndex, 3] := GuiReorientationQueueForceSingleMs3;
		BatchQueueForceSingleMs[BatchSlotIndex, 4] := GuiReorientationQueueForceSingleMs4;
		BatchQueueTriggeredMask[BatchSlotIndex] := 0;
		BatchQueueActuatedMask[BatchSlotIndex] := 0;
		BatchQueueFinishedMask[BatchSlotIndex] := (NOT BatchQueueArrayMask[BatchSlotIndex]) AND BYTE#15;
		BatchQueueExitSeen[BatchSlotIndex] := FALSE;
		BatchLastAcceptedCommit := GuiReorientationQueueCommit;
		ReorientationQueueEnqueueAck := GuiReorientationQueueSequence;
	END_IF
END_IF

IF GuiReorientationControlActive AND ((ReorientationState = 20) OR (ReorientationState = 30))
	AND (GuiReorientationResultAck <> BatchAcceptedResultAck) THEN
	IF (GuiReorientationResultAck = (BatchAcceptedResultAck + 1))
		AND (GuiReorientationResultAck <= ReorientationQueueCompletedCount) THEN
		BatchAcceptedResultAck := GuiReorientationResultAck;
	ELSE
		ReorientationFaultCode := 92; // invalid or out-of-order result acknowledgement
		ReorientationState := 92;
		ReorientationSafeLatch := TRUE;
	END_IF
END_IF

IF ReorientationQueueEnqueueAck >= BatchAcceptedResultAck THEN
	ReorientationQueueDepth := UDINT_TO_UINT(ReorientationQueueEnqueueAck - BatchAcceptedResultAck);
ELSE
	ReorientationQueueDepth := 0;
END_IF

// Record every accepted stable transition at PLC-cycle resolution for ADS diagnostics.
LightBarrierEventHistory[0] := 1;
LightBarrierEventHistory[2] := LightBarrierEventClockMs;
IF LightBarrierStable1 <> LastLightBarrier1 THEN
	LightBarrierEventCount1 := LightBarrierEventCount1 + 1;
	LightBarrierLastEventTimeMs1 := LightBarrierEventClockMs;
	LightBarrierLastEventPosition1 := StepperInternalPosition;
	LightBarrierHistorySlot := 3 + (((LightBarrierEventHistory[1] + 1) MOD 256) * 3);
	LightBarrierEventHistory[LightBarrierHistorySlot + 1] := LightBarrierEventClockMs;
	LightBarrierEventHistory[LightBarrierHistorySlot + 2] := 2 + BOOL_TO_UDINT(LightBarrierStable1);
	LightBarrierEventHistory[LightBarrierHistorySlot] := LightBarrierEventHistory[1] + 1;
	LightBarrierEventHistory[1] := LightBarrierEventHistory[LightBarrierHistorySlot];
END_IF
IF LightBarrierStable2 <> LastLightBarrier2 THEN
	LightBarrierEventCount2 := LightBarrierEventCount2 + 1;
	LightBarrierLastEventTimeMs2 := LightBarrierEventClockMs;
	LightBarrierLastEventPosition2 := StepperInternalPosition;
	LightBarrierHistorySlot := 3 + (((LightBarrierEventHistory[1] + 1) MOD 256) * 3);
	LightBarrierEventHistory[LightBarrierHistorySlot + 1] := LightBarrierEventClockMs;
	LightBarrierEventHistory[LightBarrierHistorySlot + 2] := 4 + BOOL_TO_UDINT(LightBarrierStable2);
	LightBarrierEventHistory[LightBarrierHistorySlot] := LightBarrierEventHistory[1] + 1;
	LightBarrierEventHistory[1] := LightBarrierEventHistory[LightBarrierHistorySlot];
END_IF
IF LightBarrierStable3 <> LastLightBarrier3 THEN
	LightBarrierEventCount3 := LightBarrierEventCount3 + 1;
	LightBarrierLastEventTimeMs3 := LightBarrierEventClockMs;
	LightBarrierLastEventPosition3 := StepperInternalPosition;
	LightBarrierHistorySlot := 3 + (((LightBarrierEventHistory[1] + 1) MOD 256) * 3);
	LightBarrierEventHistory[LightBarrierHistorySlot + 1] := LightBarrierEventClockMs;
	LightBarrierEventHistory[LightBarrierHistorySlot + 2] := 6 + BOOL_TO_UDINT(LightBarrierStable3);
	LightBarrierEventHistory[LightBarrierHistorySlot] := LightBarrierEventHistory[1] + 1;
	LightBarrierEventHistory[1] := LightBarrierEventHistory[LightBarrierHistorySlot];
END_IF
IF LightBarrierStable4 <> LastLightBarrier4 THEN
	LightBarrierEventCount4 := LightBarrierEventCount4 + 1;
	LightBarrierLastEventTimeMs4 := LightBarrierEventClockMs;
	LightBarrierLastEventPosition4 := StepperInternalPosition;
	LightBarrierHistorySlot := 3 + (((LightBarrierEventHistory[1] + 1) MOD 256) * 3);
	LightBarrierEventHistory[LightBarrierHistorySlot + 1] := LightBarrierEventClockMs;
	LightBarrierEventHistory[LightBarrierHistorySlot + 2] := 8 + BOOL_TO_UDINT(LightBarrierStable4);
	LightBarrierEventHistory[LightBarrierHistorySlot] := LightBarrierEventHistory[1] + 1;
	LightBarrierEventHistory[1] := LightBarrierEventHistory[LightBarrierHistorySlot];
END_IF
IF LightBarrierStable5 <> LastLightBarrier5 THEN
	LightBarrierEventCount5 := LightBarrierEventCount5 + 1;
	LightBarrierLastEventTimeMs5 := LightBarrierEventClockMs;
	LightBarrierLastEventPosition5 := StepperInternalPosition;
	LightBarrierHistorySlot := 3 + (((LightBarrierEventHistory[1] + 1) MOD 256) * 3);
	LightBarrierEventHistory[LightBarrierHistorySlot + 1] := LightBarrierEventClockMs;
	LightBarrierEventHistory[LightBarrierHistorySlot + 2] := 10 + BOOL_TO_UDINT(LightBarrierStable5);
	LightBarrierEventHistory[LightBarrierHistorySlot] := LightBarrierEventHistory[1] + 1;
	LightBarrierEventHistory[1] := LightBarrierEventHistory[LightBarrierHistorySlot];
END_IF
IF LightBarrierStable6 <> LastLightBarrier6 THEN
	LightBarrierEventCount6 := LightBarrierEventCount6 + 1;
	LightBarrierLastEventTimeMs6 := LightBarrierEventClockMs;
	LightBarrierLastEventPosition6 := StepperInternalPosition;
	LightBarrierHistorySlot := 3 + (((LightBarrierEventHistory[1] + 1) MOD 256) * 3);
	LightBarrierEventHistory[LightBarrierHistorySlot + 1] := LightBarrierEventClockMs;
	LightBarrierEventHistory[LightBarrierHistorySlot + 2] := 12 + BOOL_TO_UDINT(LightBarrierStable6);
	LightBarrierEventHistory[LightBarrierHistorySlot] := LightBarrierEventHistory[1] + 1;
	LightBarrierEventHistory[1] := LightBarrierEventHistory[LightBarrierHistorySlot];
END_IF
IF LightBarrierStable7 <> LastLightBarrier7 THEN
	LightBarrierEventCount7 := LightBarrierEventCount7 + 1;
	LightBarrierLastEventTimeMs7 := LightBarrierEventClockMs;
	LightBarrierLastEventPosition7 := StepperInternalPosition;
	LightBarrierHistorySlot := 3 + (((LightBarrierEventHistory[1] + 1) MOD 256) * 3);
	LightBarrierEventHistory[LightBarrierHistorySlot + 1] := LightBarrierEventClockMs;
	LightBarrierEventHistory[LightBarrierHistorySlot + 2] := 14 + BOOL_TO_UDINT(LightBarrierStable7);
	LightBarrierEventHistory[LightBarrierHistorySlot] := LightBarrierEventHistory[1] + 1;
	LightBarrierEventHistory[1] := LightBarrierEventHistory[LightBarrierHistorySlot];
END_IF
IF LightBarrierStable8 <> LastLightBarrier8 THEN
	LightBarrierEventCount8 := LightBarrierEventCount8 + 1;
	LightBarrierLastEventTimeMs8 := LightBarrierEventClockMs;
	LightBarrierLastEventPosition8 := StepperInternalPosition;
	LightBarrierHistorySlot := 3 + (((LightBarrierEventHistory[1] + 1) MOD 256) * 3);
	LightBarrierEventHistory[LightBarrierHistorySlot + 1] := LightBarrierEventClockMs;
	LightBarrierEventHistory[LightBarrierHistorySlot + 2] := 16 + BOOL_TO_UDINT(LightBarrierStable8);
	LightBarrierEventHistory[LightBarrierHistorySlot] := LightBarrierEventHistory[1] + 1;
	LightBarrierEventHistory[1] := LightBarrierEventHistory[LightBarrierHistorySlot];
END_IF

// Continuous part cursor. Every sensor sees sequence 1, 2, 3, ... in exactly
// that order. Odd barriers capture time; the following even barrier creates an
// immutable array job and computes its final offset delay from that same part.
BatchSensorFalling[1] := PairedFirstBarrierFalling[1];
BatchSensorFalling[2] := PairedSecondBarrierFalling[1];
BatchSensorFalling[3] := PairedFirstBarrierFalling[2];
BatchSensorFalling[4] := PairedSecondBarrierFalling[2];
BatchSensorFalling[5] := PairedFirstBarrierFalling[3];
BatchSensorFalling[6] := PairedSecondBarrierFalling[3];
BatchSensorFalling[7] := PairedFirstBarrierFalling[4];
BatchSensorFalling[8] := PairedSecondBarrierFalling[4];
BatchSensorStable[1] := LightBarrierStable1;
BatchSensorStable[2] := LightBarrierStable2;
BatchSensorStable[3] := LightBarrierStable3;
BatchSensorStable[4] := LightBarrierStable4;
BatchSensorStable[5] := LightBarrierStable5;
BatchSensorStable[6] := LightBarrierStable6;
BatchSensorStable[7] := LightBarrierStable7;
BatchSensorStable[8] := LightBarrierStable8;
BatchCurrentBarrierStableMask := BYTE#0;
IF BatchSensorStable[1] THEN BatchCurrentBarrierStableMask := BatchCurrentBarrierStableMask OR BYTE#1; END_IF
IF BatchSensorStable[2] THEN BatchCurrentBarrierStableMask := BatchCurrentBarrierStableMask OR BYTE#2; END_IF
IF BatchSensorStable[3] THEN BatchCurrentBarrierStableMask := BatchCurrentBarrierStableMask OR BYTE#4; END_IF
IF BatchSensorStable[4] THEN BatchCurrentBarrierStableMask := BatchCurrentBarrierStableMask OR BYTE#8; END_IF
IF BatchSensorStable[5] THEN BatchCurrentBarrierStableMask := BatchCurrentBarrierStableMask OR BYTE#16; END_IF
IF BatchSensorStable[6] THEN BatchCurrentBarrierStableMask := BatchCurrentBarrierStableMask OR BYTE#32; END_IF
IF BatchSensorStable[7] THEN BatchCurrentBarrierStableMask := BatchCurrentBarrierStableMask OR BYTE#64; END_IF
IF BatchSensorStable[8] THEN BatchCurrentBarrierStableMask := BatchCurrentBarrierStableMask OR BYTE#128; END_IF
BatchPairSpacingMm[1] := GuiSensorSpacing12Mm;
BatchPairSpacingMm[2] := GuiSensorSpacing34Mm;
BatchPairSpacingMm[3] := GuiSensorSpacing56Mm;
BatchPairSpacingMm[4] := GuiSensorSpacing78Mm;
BatchSensorToArraySpacingMm[1] := GuiSensor2ToArray1SpacingMm;
BatchSensorToArraySpacingMm[2] := GuiSensor4ToArray2SpacingMm;
BatchSensorToArraySpacingMm[3] := GuiSensor6ToArray3SpacingMm;
BatchSensorToArraySpacingMm[4] := GuiSensor8ToArray4SpacingMm;

IF GuiReorientationControlActive AND ((ReorientationState = 20) OR (ReorientationState = 30)) THEN
	FOR BatchLoopIndex := 1 TO 8 DO
		IF BatchSensorStable[BatchLoopIndex] THEN
			BatchSensorNeedsClear[BatchLoopIndex] := FALSE;
		END_IF
		IF BatchSensorFalling[BatchLoopIndex] THEN
			ReorientationFaultSensor := INT_TO_UINT(BatchLoopIndex);
			ReorientationFaultExpectedSequence := BatchNextSensorSequence[BatchLoopIndex];
			ReorientationFaultPreviousSequence := 0;
			ReorientationFaultQueueAck := ReorientationQueueEnqueueAck;
			ReorientationFaultBarrierStableMask := BatchCurrentBarrierStableMask;
			IF BatchSensorNeedsClear[BatchLoopIndex] THEN
				ReorientationFaultDetail := 1;
				ReorientationFaultQueueSlotSequence := 0;
				// Diagnostic mode: reject the ambiguous edge but keep production
				// running. Never advance a cursor or trigger a nozzle from it.
				ReorientationWarningCode := 3;
				ReorientationWarningSensor := INT_TO_UINT(BatchLoopIndex);
				ReorientationWarningSequence := BatchNextSensorSequence[BatchLoopIndex];
				ReorientationWarningPreviousSequence := 0;
				ReorientationWarningSkippedBarrierMask := BYTE#0;
				ReorientationWarningCounter := ReorientationWarningCounter + 1;
				IF (BatchLoopIndex MOD 2) = 1 THEN
					BatchJobIndex := (BatchLoopIndex + 1) / 2;
					PairedFirstBarrierLocked[BatchJobIndex] := TRUE;
					PairedFirstBarrierLockStartMs[BatchJobIndex] := LightBarrierEventClockMs;
					PairedSecondBarrierLocked[BatchJobIndex] := FALSE;
				ELSE
					BatchJobIndex := BatchLoopIndex / 2;
					PairedSecondBarrierLocked[BatchJobIndex] := TRUE;
					PairedSecondBarrierLockStartMs[BatchJobIndex] := LightBarrierEventClockMs;
					PairedFirstBarrierLocked[BatchJobIndex] := FALSE;
				END_IF
			ELSE
				BatchSensorNeedsClear[BatchLoopIndex] := TRUE;
				BatchSlotIndex := UDINT_TO_INT((BatchNextSensorSequence[BatchLoopIndex] - 1) MOD 128);
				// A normal TwinCAT AND does not guarantee short-circuit evaluation.
				// Never form BatchSensorSequence[0] while processing sensor 1.
				BatchSensorOrderInvalid := FALSE;
				BatchCanResyncSkippedSensors := FALSE;
				BatchCurrentFlightConfirmed := FALSE;
				BatchIgnoreAirborneDuplicate := FALSE;
				BatchLastRequiredSensor := 0;
				BatchLastRequiredArrayMask := BYTE#0;
				BatchPreviousLastRequiredSensor := 0;
				BatchPreviousLastRequiredArrayMask := BYTE#0;
				IF BatchLoopIndex > 1 THEN
					ReorientationFaultPreviousSequence := BatchSensorSequence[BatchLoopIndex - 1];
					BatchSensorOrderInvalid :=
						BatchSensorSequence[BatchLoopIndex - 1] < BatchNextSensorSequence[BatchLoopIndex];
					// The highest enabled array defines the final sensor pair that
					// remains timing/actuation-critical for this queued part.
					IF (BatchQueueArrayMask[BatchSlotIndex] AND BYTE#8) <> BYTE#0 THEN
						BatchLastRequiredSensor := 8;
						BatchLastRequiredArrayMask := BYTE#8;
					ELSIF (BatchQueueArrayMask[BatchSlotIndex] AND BYTE#4) <> BYTE#0 THEN
						BatchLastRequiredSensor := 6;
						BatchLastRequiredArrayMask := BYTE#4;
					ELSIF (BatchQueueArrayMask[BatchSlotIndex] AND BYTE#2) <> BYTE#0 THEN
						BatchLastRequiredSensor := 4;
						BatchLastRequiredArrayMask := BYTE#2;
					ELSIF (BatchQueueArrayMask[BatchSlotIndex] AND BYTE#1) <> BYTE#0 THEN
						BatchLastRequiredSensor := 2;
						BatchLastRequiredArrayMask := BYTE#1;
					END_IF
					BatchCurrentFlightConfirmed :=
						(BatchLastRequiredArrayMask <> BYTE#0)
						AND ((BatchQueueActuatedMask[BatchSlotIndex]
							AND BatchLastRequiredArrayMask) <> BYTE#0);
					BatchCanResyncSkippedSensors := BatchSensorOrderInvalid
						AND ((BatchLoopIndex - 1) > BatchLastRequiredSensor)
						AND BatchCurrentFlightConfirmed;

